(* CoDeSys 2.3 export: PALETIZER.EXP *)

(* Data type in EPT Lib/Achsen/BECKHOFF *)
TYPE struct_eccoe_sdo :
STRUCT
	s_ec_slave_net_id 		: T_AmsNetId := '';
	ui16_slave_addr 			: UINT := 0; (* Address of the slave device.*)
	i8_sub_index 				: BYTE := 0; (* CANopen Sdo subindex.*)
	w_index 					: WORD := 16#00; (* CANopen Sdo index.*)
	dw_p_source_buffer 		: DWORD := 16#0000; (* Contains the address of the buffer containing the data to be send. *)
	dw_p_destination_buffer	: DWORD := 16#0000; (* Contains the address of the buffer for the received data. *)
	ui32_buffer_length 			: UDINT := 0; (* Contains the max. number of bytes to be received. *)
	ui32_value 				: UDINT := 0; (* variable to be written to the CoE Object *)
	ui16_value 				: UINT := 0; (* variable to be written to the CoE Object *)
	byte_value 				: BYTE := 16#00; (* variable to be written to the CoE Object *)
	bool_value 				: BOOL := FALSE; (* variable to be written to the CoE Object *)
END_STRUCT
END_TYPE

(* Data type in EPT Lib/Achsen/EL72x1 *)
TYPE enum_ModeOfOperation :
	(
	CSP			:=	8,	(*cyclic synchronous position*)
	CSV			:=	9,	(*cyclic synchronous velocity*)
	CST			:=	10,	(*cyclic synchronous torque*)
	CSTCA		:=	11	(*cyclic synchronous torque with commutation angle*)
	);
END_TYPE

(* Data type in EPT Lib/Achsen/EL72x1 *)
TYPE st_config_axis :
STRUCT
	Description				:STRING;
	InstName				:STRING;
	Aktiv					:BOOL;
	Skalierfaktor				:LREAL;
	Bit_Geber				:INT;
	Getriebefaktor			:LREAL;
	Modulo					:BOOL:=TRUE;
	Pos_Faktor				:LREAL;						(*Weg bei einer Motorumdrehung in mm*)
	ModeOfOperation			:enum_ModeOfOperation:=CSP;
	maxRpm					:INT;				(*Maximale Drehzahl des Motor*)
(*nur für Coe-Online 7010.03 (CSP) position mode*)

	RampTime				:TIME;				(*Baustelle*)(*Beschleunigungszeit und Bremsrampe*)
	PosDiffControl_on			:BOOL;				(*Baustelle*)
	max_PosDiff				:LREAL;				(*Baustelle*)
	UeberlaufControl_on		:BOOL;
	Torque_Limit				:INT;				(*bei 0 ausgeschaltet*)(* Baustelle*)
	SW_Limit_on				:BOOL;
	SW_Limit_min			:LREAL;
	SW_Limit_max			:LREAL;
	lr_kp 					:LREAL := 800;
	lr_ki 						:LREAL := 100.0;
	lr_kd 					:LREAL := 50;
END_STRUCT
END_TYPE

(* Data type in EPT Lib/Achsen/EL72x1 *)
TYPE st_ctrl_Axis :
STRUCT
	in		: st_ctrl_in_axis;
	out		: st_ctrl_out_axis;
END_STRUCT
END_TYPE

(* Data type in EPT Lib/Achsen/EL72x1 *)
TYPE st_ctrl_in_axis :
STRUCT
	Position					:LREAL;

(*Bit 0*) Ready_to_switch_on	:BOOL;
(*Bit 1*) Switched_on			:BOOL;
(*Bit 2*) Operation_enabled		:BOOL;
(*Bit 3*) Fault					:BOOL;
(*Bit 4 : reserved*)
(*Bit 5 : reserved*)
(*Bit 6*) Switch_on_disabled		:BOOL;
(*Bit 7*) Warning				:BOOL;
(*Bit 8 + 9 : reserved*)
(*Bit 10*) TxPDOToggle		:BOOL; (*An-/Abwahl über 0x8010:01[} 136]*)
(*Bit 11*) Internal_Limit_active	:BOOL;
(*Bit 12*) Target_value_ignored	:BOOL;
(*Bit 13 - 15 : reserved*)

	Velocity				:LREAL;
	Following_Error		:LREAL;

END_STRUCT
END_TYPE

(* Data type in EPT Lib/Achsen/EL72x1 *)
TYPE st_ctrl_out_axis :
STRUCT
	Target_Position		:LREAL;
	Tearget_Velocity		:DINT;

(*Bit 0*)	Switch_on					:BOOL;
(*Bit 1*)	Enable_voltage		:BOOL;
(*Bit 2	*)Shutdown					:BOOL;
(*Bit 3*)	Enable_operation	:BOOL;
(*Bit 4 - 6 : reserved*)
(*Bit 7*)	Fault_reset				:BOOL;
(*Bit 8 - 15 : reserved*)

END_STRUCT
END_TYPE

(* Data type in EPT Lib/Achsen/EL72x1 *)
TYPE st_fb_axis :
STRUCT
	ton_uez			:TON;
	ton_uez_velo	:TON;
	ton_quitt		:TON;
	ton_aufPos		:TON;
	ton_Busy		:TON;


	r_trig_stop		: R_TRIG;
	r_trig_quitt	: R_TRIG;
	r_trig_reset	: R_TRIG;
	r_trig_jogP		: R_TRIG;
	r_trig_jogM		: R_TRIG;
	r_trig_MoveP	: R_TRIG;
	r_trig_MoveM	: R_TRIG;
	r_trig_MotorOn	: R_TRIG;
	r_trig_MoveAbs	: R_TRIG;

	r_trig_teach		: R_TRIG;
	r_trig_kont			: R_TRIG;
	r_trig_ink_10		: R_TRIG;
	r_trig_ink_100		: R_TRIG;
	r_trig_ink_1000		: R_TRIG;
	r_trig_ink_var		: R_TRIG;
	r_trig_Auto			: R_TRIG;
	r_trig_Hand			: R_TRIG;
END_STRUCT
END_TYPE

(* Data type in EPT Lib/Achsen/EL72x1 *)
TYPE st_Help_axis :
STRUCT
	b_init				:BOOL;
	b_init2				:BOOL;
	b_ToggleHelp		:BOOL;

	b_Pos_nr_Empty		:ARRAY [-1..NO_OF_POS_AXIS] OF BOOL;
	PosNr				:INT:=1;
	Pos					:LREAL;

END_STRUCT
END_TYPE

(* Data type in EPT Lib/Achsen/EL72x1 *)
TYPE st_PID_axis :
STRUCT
	lr_Override			:LREAL;

	lr_delta				: LREAL := 0.0;
	lr_delta_alt			: LREAL := 0.0;
	lr_delta_dif			: LREAL := 0.0;

	lr_current_p			: LREAL := 0.0;
	lr_current_i			: LREAL := 0.0;
	lr_current_d			: LREAL := 0.0;

	lr_current_v			: LREAL := 0.0;
	lr_tmp				: LREAL := 0.0;

	lr_delta_targetpos	: LREAL := 0.0;
	lr_targetpos_alt		: LREAL := 0.0;

END_STRUCT
END_TYPE

(* Data type in EPT Lib/Achsen/EL72x1 *)
TYPE st_Pos :
STRUCT
	Description		: STRING;
	Pos	 			: LREAL;
END_STRUCT
END_TYPE

(* Data type in EPT Lib/Achsen/EL72x1 *)
TYPE st_Pos_axis :
STRUCT
	ist					:REAL;
	soll					:REAL;
	r_18bit				:REAL;
	r_20bit				:REAL;
	r_32bit				:REAL;

	lr_DiffPuls			:LREAL := 0.0;
	lr_DiffVelo			:LREAL := 0.0;
	lr_MaxDiff			:LREAL := 0.0;

	(*Überlauf*)
	lr_akt_alt				:LREAL;
	lr_delta_ueberlauf		:LREAL;
	i32_count_ueberlauf	:DINT;
	lr_Uebrlauf_DistOne	:LREAL;
	lr_Uebrlauf_Dist		:LREAL;

	(*Singelturn*)
	lr_ModuloPosInc		:LREAL;
	lr_ModuloHelp		:LREAL;
	lr_ModuloHelp2		:LREAL;
	i16_ModuloHelp		:INT;
	lr_ModuloCount		:LREAL;

	(*Multiturn*)
	lr_Pos				:LREAL;
	lr_Target				:LREAL;
	lr_Mod				:LREAL;

	lr_Offset_Ink			:LREAL;
	i32_Offset_Ink			:UDINT;

END_STRUCT
END_TYPE

(* Data type in EPT Lib/Achsen/EL72x1 *)
TYPE st_sdo :
STRUCT
	fb_ec_coe_sdo_write_ex		: FB_EcCoESdoWriteEx;
	fb_ec_coe_sdo_read_ex		: FB_EcCoESdoReadEx;

(*	st_eccoe_sdo				:struct_eccoe_sdo;*)

	s_SlaveNetId 			: T_AmsNetId := '';
	ui16_SlaveAddr 			: UINT := 0;			 (* Address of the slave device.*)
	i8_SubIndex 			: BYTE := 0;			 (* CANopen Sdo subindex.*)
	w_Index 				: WORD := 16#00;	 (* CANopen Sdo index.*)

	acObjectData				:ARRAY[0..MAX_STRING_LENGTH] OF BYTE;

END_STRUCT
END_TYPE

(* Data type in EPT Lib/Achsen/EL72x1 *)
TYPE st_sm_axis :
STRUCT
	sm_timeout			:BOOL;
	sm_Error_Klemme	:BOOL;
	sm_Error_Warnung	:BOOL;
	sm_PosDiff			:BOOL;
	sm_Check_Velo		:BOOL;
	sm_SW_Limit			:BOOL;
	sm_fehler_daten_schreiben:BOOL;
	sm_connect			:BOOL;
	sm_Ueberlauf		:BOOL;
	sm_Torque_zu_gross	:BOOL;
	sm_NotausNok		:BOOL;
	sm_Move				:BOOL;
END_STRUCT
END_TYPE

(* Data type in EPT Lib/Achsen/EL72x1 *)
TYPE st_Velo_axis :
STRUCT
	maxRpmNachGertiebe	:LREAL;	(*Maximale Drehzahl nach Getriebe*)
	maxLinear		:LREAL;	(*Maximale Geschwindigkeit in mm/min*)
	maxRpm				:LREAL;	(*in U/min oder in mm/min*)
	Vorgabe_Velo_rpm	:LREAL;	(*in U/min*)
	sollRpm				:LREAL;	(*in U/min*)
	soll					:LREAL;
	ist				:LREAL;
	dif				:LREAL;
	Faktor			:LREAL;

END_STRUCT
END_TYPE

(* Data type in EPT Lib/Achsen/EL72x1 *)
TYPE st_Visu_axis :
STRUCT
	Einheit_pos			:STRING(10);
	Einheit_velo			:STRING(10);

	BtnReset			: sButtonVisu;
	BtnStop				: sButtonVisu;
	BtnJogP			: sButtonVisu;
	BtnJogM			: sButtonVisu;
	BtnMotorOn			: sButtonVisu;
	BtnMoveAbs		: sButtonVisu;
	BtnTeach			: sButtonVisu;

	PosNr				:INT:=1;
	Poslist				:BOOL;

	Control				:BOOL;
	b_kont				:BOOL;
	b_ink_10			:BOOL;		(*in µm*)
	b_ink_100			:BOOL;		(*in µm*)
	b_ink_1000			:BOOL;		(*in µm*)
	b_ink_var			:BOOL;		(*in mm variabel *)
	lr_ink_var			:LREAL:=10;

	b_Pos_nr			:ARRAY [-1..NO_OF_POS_AXIS] OF BOOL;
	b_PosNr			:BOOL;
END_STRUCT
END_TYPE

(* Data type in EPT Lib/Allgemeine Kontrollstrukturen Objekte *)
TYPE enum_step_nr :
	(
	INIT_OBJ := 0,
	INIT := 10,
	BEREIT := 100,
	HALT := 970,
	STOP := 980,
	FEHLER := 1000,
	INAKTIV:=2010
	);
END_TYPE

(* Data type in EPT Lib/Allgemeine Kontrollstrukturen Objekte *)
TYPE struct_config :
STRUCT
	str_instanz_name					: STRING(48) := '';
	str_beschreibung					: STRING(50) := '';
	b_station_aktiv					: BOOL := FALSE;
	b_station_in_simulation				: BOOL := FALSE;
	i16_meld_startindex				: INT := 0;
	b_config_fertig					: BOOL := FALSE;
END_STRUCT
END_TYPE

(* Data type in EPT Lib/Allgemeine Kontrollstrukturen Objekte *)
TYPE struct_ctrl :
STRUCT
	in		: struct_ctrl_in;
	out		: struct_ctrl_out;
END_STRUCT
END_TYPE

(* Data type in EPT Lib/Allgemeine Kontrollstrukturen Objekte *)
TYPE struct_ctrl_in :
STRUCT
	b_quitt						: BOOL := FALSE;
	b_stop 						: BOOL := FALSE;
         b_halt		  	 			: BOOL := FALSE;
         b_definierter_halt  	 			: BOOL := FALSE;
	b_init 						: BOOL := FALSE;
	b_init_2 						: BOOL := FALSE;
         b_preinit                				: BOOL := FALSE;
	b_start						: BOOL := FALSE;
	b_start_2						: BOOL := FALSE;
	b_gutteil_produziert 			: BOOL := FALSE;
	b_schlechtteil_produziert 		: BOOL := FALSE;
	b_start_lesen					: BOOL := FALSE;
	b_start_schreiben				: BOOL := FALSE;
	b_schutzhaube_ab			: BOOL := FALSE;
	b_schutzhaube_auf			: BOOL := FALSE;
	b_nachtabschaltung			: BOOL := FALSE;
	b_gehe_step_ibn				: BOOL := FALSE;
	b_ibn_start					: BOOL := FALSE;
	b_freigabe					: BOOL := FALSE;
END_STRUCT
END_TYPE

(* Data type in EPT Lib/Allgemeine Kontrollstrukturen Objekte *)
TYPE struct_ctrl_out :
STRUCT
	b_bereit 						: BOOL := FALSE;
	b_bereit_2					: BOOL := FALSE;
         b_prebereit               			: BOOL := FALSE;
	b_fehler 						: BOOL := FALSE;
	b_fertig						: BOOL := FALSE;
	b_fertig_2					: BOOL := FALSE;
	b_bandende					: BOOL := FALSE;
	b_kontroller_start				: BOOL := FALSE;
	b_gestoppt					: BOOL := FALSE;
	b_angehalten					: BOOL := FALSE;
	b_haube_oeffnen				: BOOL := FALSE;
	b_nachtabschaltung			: BOOL := FALSE;
	b_einzelfertigung				: BOOL := FALSE;
	b_busy						: BOOL := FALSE;
 st_takt_Time : STRING;
END_STRUCT
END_TYPE

(* Data type in EPT Lib/Allgemeine Kontrollstrukturen Objekte *)
TYPE struct_objekt :
STRUCT
	st_config		: struct_config;
	st_ctrl		: struct_ctrl;
END_STRUCT
END_TYPE

(* Data type in EPT Lib/Hydra *)
TYPE enum_StatusId :
	(

		(*
		M_S = Maschinenstörung,
		W_S = Werkzeugstörung,
		P_S = Peripheriestörung,
		AOI_S = Kamerastörung,
		M_W = Maschinenwartung,
		W_W = Werkzeugwartung,
		A_U = Ablaufunterbrechung
		*)


		_PRODUKTION := 1,
		_Nachtabschaltung_STOP := 199,
		_S_Quittiert := 290,
		_A_U_Steuerung_Aus := 299,
		_A_U_Auftrag_voll := 300,
		_M_S_Haube_Einzug := 301,
		_A_U_Trennstelle := 303,
		_A_U_Spule_voll := 304,
		_M_S_Haubenschaltleiste := 305,
		_M_S_Haube_Bandauslauf := 306,
		_M_S_Klappe_hinten := 307,
		_M_S_Klappe_links := 308,
		_M_S_Klappe_rechts := 309,
		_M_S_Klappe_vorne := 310,
		_M_S_Temp_Schaltschrank := 311,
		_M_S_Temp_Haubenmotor := 312,
		_M_S_Temp_Haubenluefter := 313,
		_M_S_Bandoeler_Fuellstand := 314,
		_M_S_Bandoeler := 315,
		_M_W_Pressenkopf := 316,
		_M_W_Zahnriemen := 317,
		_M_W_Wartungseinheit := 318,
		_M_W_Bandeinzug := 319,
		_M_W_Werkzeug := 320,
		_M_S_Drehgeber := 321,
		_M_S_Hauptantriebsmotor := 322,
		_M_S_Abfallbehaelter := 323,
		_W_S_Bandaufgestellt := 325,
		_W_S_Parallelschnitt := 326,
		_W_S_Gesamtschnitt_o := 327,
		_W_S_Gesamtschnitt_u := 328,
		_W_S_Dyn_Schnittueberw_eins := 329,
		_W_S_Dyn_Schnittueberw_zwei := 331,
		_W_S_Faengerueberw_eins := 332,
		_W_S_Faengerueberw_zwei := 333,
		_W_S_Faengerueberw_drei := 334,
		_W_S_Faengerueberw_vier := 335,
		_W_S_Position_Wkz := 336,
		_W_S_Pfostenabfrage := 337,
		_W_S_Tcom_eins := 338,
		_W_S_Tcom_zwei := 339,
		_W_S_Bandschneideueberwachung := 340,
		_W_S_Pinabstanzueberwachung := 341,
		_AOI_S_Kamera :=343,
		_P_S_Aufhaspel := 350,
		_P_S_Abhaspel := 351,
		_M_S_Not_Halt := 352,
		_M_S_Auffahrsicherung := 353,
		_Trennstelle := 809,
		_Maschine_STOP :=843,
		_Peripherie_STOP := 844,
		_Stoerung_Lasertriangulation := 870,
		_Stoerung_Bsh_Zellen := 871,
		_Maschinenstoerung := 884,
		_Peripheriestoerung := 885,
		_WERKZEUGSTOERUNG := 886,
		 _Kamerastoerung := 887,
		_HV_Stoerung := 888,
		_Schichtfrei := 999

);

END_TYPE

(* Data type in EPT Lib/Hydra *)
TYPE struct_Hydra :
STRUCT
	s_Start_Time	: STRING(20) := '01.01.1970 00:00:00';	(* TT.MM.JJJJ HH:MM:SS *)
	i_Counter		: ARRAY[1..104] OF DINT;	(* alle Zähler 4-stellig *)
	b_Input		: ARRAY[1..128] OF BOOL:=128(FALSE);
END_STRUCT
END_TYPE

(* Data type in EPT Lib/Hydra *)
TYPE struct_Hydra8 :
STRUCT
	iCounter		: ARRAY[1..20] OF DINT;	(* alle Zähler 4-stellig *)
	bStatus		: ARRAY[1..999] OF BOOL:=999(FALSE);	(* TRUE wenn Status aktiv ist *)
END_STRUCT
END_TYPE

(* Data type in EPT Lib/sDatensatz/sTypeDaten *)
TYPE sData_b :
STRUCT

	Description					: STRING(50); 	(* Beschreibung *)
	b								: BOOL; 		(* Wert *)

END_STRUCT
END_TYPE

(* Data type in EPT Lib/sDatensatz/sTypeDaten *)
TYPE sData_byte :
STRUCT

	Description					: STRING(50); 	(* Beschreibung *)
	BYT								: BYTE; 			(* Wert *)
	Unit				   			: STRING(20);	(* Einheit *)

END_STRUCT
END_TYPE

(* Data type in EPT Lib/sDatensatz/sTypeDaten *)
TYPE sData_i16 :
STRUCT

	Description					: STRING(50); 	(* Beschreibung *)
	i16								: INT; 			(* Wert *)
	Unit				   			: STRING(20);	(* Einheit *)

END_STRUCT
END_TYPE

(* Data type in EPT Lib/sDatensatz/sTypeDaten *)
TYPE sData_i32 :
STRUCT

	Description		: STRING(50); 	(* Beschreibung *)
	i32					: DINT; 		(* Wert *)
	Unit				: STRING(20);	(* Einheit *)

END_STRUCT
END_TYPE

(* Data type in EPT Lib/sDatensatz/sTypeDaten *)
TYPE sData_lr :
STRUCT

	Description		: STRING(50); 	(* Beschreibung *)
	lr					: LREAL; 			(* Wert *)
	Unit		   		: STRING(20);	 	(* Einheit *)

END_STRUCT
END_TYPE

(* Data type in EPT Lib/sDatensatz/sTypeDaten *)
TYPE sData_Str :
STRUCT

	Description				: STRING(50); 	(* Beschreibung *)
	str							: STRING(50); 	(* Text *)

END_STRUCT
END_TYPE

(* Data type in EPT Lib/sDatensatz/sTypeDaten *)
TYPE sData_ui32 :
STRUCT

	Description			: STRING(50); 	(* Beschreibung *)
	i32						: UDINT; 		(* Wert *)
	Unit					: STRING(20);	(* Einheit *)

END_STRUCT
END_TYPE

(* Data type in sStation/MainMenue *)
TYPE sMainMenue:
STRUCT
	BtnMainMenue					:sButtonVisu_Tree;
	BtnManual						:sButtonVisu_Tree;
	BtnManual_ST00_0				:sButtonVisu_Tree;	(*Allgemein*)
		BtnManual_ST00_1			:sButtonVisu_Tree;	(*Türen und Not-Halt*)
		BtnManual_ST00_2			:sButtonVisu_Tree;	(*Flügelkamera*)
	BtnManual_ST02_0				:sButtonVisu_Tree;	(*Rundtisch*)
	BtnManual_ST03_0				:sButtonVisu_Tree;	(*Roboter*)
			BtnManual_ST03_xx		:sButtonVisu_Tree;	(*Rüstsatz Seite1*)
			BtnManual_ST03_xx_2	:sButtonVisu_Tree;	(*Rüstsatz Seite2*)
	BtnManual_ST08_0				:sButtonVisu_Tree;
		BtnManual_ST08_1			:sButtonVisu_Tree;	(*Blisterzuführung*)
		BtnManual_ST08_2			:sButtonVisu_Tree;	(*Abstapeln*)
		BtnManual_ST08_3			:sButtonVisu_Tree;	(*Bandstrecke*)
		BtnManual_ST08_4			:sButtonVisu_Tree;	(*Aufstapeln*)


	BtnTD							:sButtonVisu_Tree;
	BtnTD01_Edit					:sButtonVisu_Tree;
	BtnTD02_Edit					:sButtonVisu_Tree;

	BtnMP_Main					:sButtonVisu_Tree;
	BtnMP_ST1						:sButtonVisu_Tree;
	BtnMP_ST2						:sButtonVisu_Tree;
	BtnMP_Date					:sButtonVisu_Tree;
	BtnMP_Service					:sButtonVisu_Tree;

	BtnSystem						:sButtonVisu_Tree;
		Btn_ErrorLog				:sButtonVisu_Tree;
		Btn_ErrorList				:sButtonVisu_Tree;
		Btn_Gst						:sButtonVisu_Tree;
		Btn_Step_Diag				:sButtonVisu_Tree;
		Btn_Lng					:sButtonVisu_Tree;

		Btn_VisuBeenden			:sButtonVisu_Tree;
END_STRUCT
END_TYPE

(* Data type in sStation/sMachineParameter/Service *)
TYPE eService_Type :
	(
	BETRIEBSSTUNDEN			:=	0,
	STUNDEN			:=	1,
	TAGE				:=	2,
	COUNTER			:=	3
	);
END_TYPE

(* Data type in sStation/sMachineParameter/Service *)
TYPE sMachParaService :
STRUCT
	visu			: ARRAY[0..15] OF struct_visu_service;
	daten			: ARRAY[0..15] OF struct_daten_service;
	betriebssekundenzaehler	:UDINT;
END_STRUCT
END_TYPE

(* Data type in sStation/sMachineParameter/Service *)
TYPE struct_daten_service :
STRUCT
	Name			: STRING(255);
	Default_Value	: LREAL;
	Current_Value	: LREAL;
	Warning_Value	: LREAL;
	Warning_reached	: BOOL:= FALSE;
	Default_reached	: BOOL:= FALSE;
	Type_Service	: eService_Type;
	Unit				: STRING(20);
	Starttag			: INT := 0;
	Startstunden	: LREAL := 0;
	StartBetriebsStd	: LREAL := 0;
END_STRUCT
END_TYPE

(* Data type in sStation/sMachineParameter/Service *)
TYPE struct_visu_service :
STRUCT
	BtnReset			: sButtonVisu;
	BtnStart			: sButtonVisu;
	BtnType			: sButtonVisu;
	Current_Value	 : STRING(20);
	Current_Value_Color	: DINT;

END_STRUCT
END_TYPE

(* Data type in sStation/sMachineParameter *)
TYPE sMachineParameterHandling :
STRUCT
(* ST01 *)
	Dummy:BOOL;
(* ST02 *)

(* ST03 *)

(* ST04 *)

(* ST05 *)
END_STRUCT
END_TYPE

(* Data type in sStation/sMachineParameter *)
TYPE sMachPara :
STRUCT
	sLastTDfile							: STRING;
	ShiftData							: sMP_ShiftHandler;
	ST00: sMachParaST00; (*Instancename is Filename in Typedata Folder*)
	ST02: sMachParaST02; (*Instancename is Filename in Typedata Folder*)
	ST03: sMachParaST03; (*Instancename is Filename in Typedata Folder*)
	ST08: sMachParaST08; (*Instancename is Filename in Typedata Folder*)
	Visu:	sMachineParameterHandling; (* Object Collection for Parameterhandling in Visu - e.g. Buttons - Called in System/VisuInterface/MachParaHandling  *)
END_STRUCT
END_TYPE

(* Data type in sStation/sMachineParameter *)
TYPE sMachParaST00 :
STRUCT
	Override					:	DINT :=10;
	OverrideForHoming	:	DINT :=5;
	MaxLogInTime				: DINT  := 0;
	Sprache    					: STRING(10);

	ActPartNo			: DINT; (*laufende Nr. für Laser-String*)

	IFMCameraActive			: BOOL := TRUE;
	IFMCameraActiveText		:STRING :='ON';

	Cam_NoOfErrors		: DINT := 1;

(* -----------------------------------------------------------------------------------------
		Sollwerte
  ----------------------------------------------------------------------------------------- *)

	PartsToProduce					: DINT;		(* Sollstückzahl *)
	PartsToProduceOffset		: DINT;		(* Korrenkturwert auf Sollstückzahl *)

 	PartsNokInSeriesAllowed : DINT := 0;		(* max. Fehler in Folge *)

	PartsNokPerSubset				: DINT :=0;		(* max. erlaubete n.i.O. Teileanzahl pro Untermenge *)
	PartsNokSubsetSize			: DINT :=100;		(* Untermengengröße *)

(* -----------------------------------------------------------------------------------------
		Istwerte
  ----------------------------------------------------------------------------------------- *)

	PartsInserted						: DINT;		(* Teile aufgesetzt in ST01 *)
	PartsNokTotal						: DINT;		(* Teile n.i.O. gesamt *)
	PartsOkTotal						: DINT;		(* Teile i.O. gesamt, eingesetzt in Blister/Tube *)
	PartsRemaining					: DINT;		(* Teile noch zu produzieren (PartsToProduce + PartsToProduceOffset + PartsNokTotal - PartsInserted) *)

	PartsNokTotalNoReset		: DINT;		(* Teile n.i.O. gesamt *)
	PartsOkTotalNoReset			: DINT;		(* Teile i.O. gesamt, eingesetzt in Blister/Tube *)

	LAN_no						: sData_i16:=(Description:='LAN_no', Unit:='no');
END_STRUCT
END_TYPE

(* Data type in sStation/sMachineParameter *)
TYPE sMachParaST02 :
STRUCT
	Override_Band				:	DINT :=10;

	RunTableEmpty 			: DINT := 5; (*Time in sec. *)
	IFMPos					: LREAL;
	IFMPosDummy			: LREAL;
	TableData				: ARRAY [1..NO_OF_NEST] OF sStationData;
	CamOn					: BOOL;
	CamNoOfErrors			: DINT := 1;
	CamNoOfErrorsPercent	: DINT := 1;
	DummyPruefung_93pol	: BOOL;
  	Dummy_test_Result  	: ARRAY [1..12] OF BOOL;
	NoOfDummys			: DINT := 6;
	SensopartIPAdress		: STRING(15);
	SensopartIPAdress2		: STRING(15);
	SensopartEthernet		: BOOL;

END_STRUCT
END_TYPE

(* Data type in sStation/sMachineParameter *)
TYPE sMachParaST03 :
STRUCT

	WpcInStackFilled		: BOOL;

	ActualPartsInPallet 		: DINT; (* Counter *)

	NoOfBlisterInStackerOut	: DINT; (* Counter *)

	ActualPartsOnBuffer 		: DINT; (* Counter *)

	ResetBuffer             : BOOL;
	(* Inputvariablen *)
	PartsInPallet	      	   : DINT; (* Max No Of Parts in Buffer *)

	NoOfTestParts				:	DINT;

	FrontCamOn			: BOOL;
	BackCamOn			: BOOL;
	CamNoOfErrors			: DINT := 1;
	CamNoOfErrorsPercent	: DINT := 1;

	RobotIPAdress			: STRING(15);
	BandMoveP				:BOOL;
	SGM_3621		: BOOL;

	BeltMotorCheckPartActive          : BOOL;

	RoboterColisionActivated	 :BOOL;

	CamOn					: ARRAY [1..2] OF BOOL;		(*Sensopart Kamera*)
	SensopartIPAdress		: ARRAY [1..2] OF STRING(15);

	CamOn_KYE				: BOOL;			(*Keyence Kamera*)
	CamNoOfErrors_KYE		: DINT := 1;
	CamNoOfErrorsPercent_KYE: DINT := 1;

END_STRUCT
END_TYPE

(* Data type in sStation/sMachineParameter *)
TYPE sMachParaST08 :
STRUCT
	NoOfBlisterInStackerOut			: DINT; (* Counter *)

	StapelMotor								: BOOL;
	PosOffsetAufstapeln	 			: st_Pos;
	PosOffsetAbstapeln	 			: st_Pos;
	Override_Aufstapeln				: DINT :=10;
	Override_Abstapeln				: DINT :=10;
	Traystapel_schieben 			: BOOL:=TRUE;
	Trayzufuhr_Verlaengerung		: BOOL:=TRUE;
	TrayAushebenMotor				: BOOL;
	PosOffsetTrayAusheben 			: st_Pos;
	Override_TrayAusheben			: DINT :=10;

END_STRUCT
END_TYPE

(* Data type in sStation/sPersistent *)
TYPE sPersDaten :
STRUCT

	i_DayOfYearAutoCheckIn	:DINT;

END_STRUCT
END_TYPE

(* Data type in sStation/sTurnTable *)
TYPE sProcessData :
STRUCT

	Nest_Nr			: DINT;
	Part				: BOOL;
	Result 			: DINT;					(*   0 = Teil noch nicht bearbeitet bzw. Nest leer*)
											(*   1 =  Oberseite OK*)
											(*  11 = Oberseite und Unterseite OK*)
											(*  99 = Teil ist NOK	*)
END_STRUCT
END_TYPE

(* Data type in sStation/sTurnTable *)
TYPE sStationData :
STRUCT
	Description				: STRING:='';
	HomePos				: BOOL;
	Activated				: BOOL := TRUE; (* Station Deactivated *)
	CycleTime				: DINT;

	ProcessData			: sProcessData; (*is shifted when Table turns*)
END_STRUCT
END_TYPE

(* Data type in sStation/sTypedata *)
TYPE sTypeData :
STRUCT
	(* allegmeine Typinfos *)
	ArtNo					: STRING(30); (* interne Kundenartikelnummer *)
	TypeName				: STRING(30); (* xml-Dateiname *)
	TypeDescription			: STRING(30); (* Typbeschreibung optional *)

	(* Typmerkmale *)
	TypeCode				: STRING(5); (* Typkennung z.B. P310 *)

	Override_Band			: INT:=20; (* *)
	Override_Robi			: INT:=20; (* *)

	PosAbstapeln	 		: ARRAY [1..NO_OF_POS_AXIS] OF st_Pos;	(*	1=unten, 2= mitte, 3=oben*)
	PosAufstapeln	 		: ARRAY [1..NO_OF_POS_AXIS] OF st_Pos;	(*	1=unten, 2= mitte, 3=oben*)
	PosTrayAusheben	 		: ARRAY [1..NO_OF_POS_AXIS] OF st_Pos;	(*	1=unten, 2=oben*)

	TestpartBilister		: BOOL;
	DistIso					: LREAL;

	IFM_Positon_Dummy 		: LREAL ;
	SensopartErgebnis			: STRING(15); (*Ergebnis Sensopart Kamera*)
	Sensopart2Ergebnis			: STRING(15); (*Ergebnis Sensopart Kamera*)
	NoOfPalletsPerStack		: DINT:=1;

	(*Aus Load Info*)
	RobotOffset				: DINT;

	PartsInBlisterInlet		: DINT; (* Anzahl Teile pro Blister Einlauf *)
	PartsInRoboGripper		: DINT:=1; (* Anzahl Teile pro Robi Greifer *)

	IFM_CamProgNo			: BYTE;
	Sensopart_CamProgNo		: BYTE;
	Sensopart2_CamProgNo		: BYTE;
	Keyence_CamProgNo		: BYTE;

END_STRUCT
END_TYPE

(* Data type in sStation/sUserList *)
TYPE sUserList :
STRUCT
  	UserList							:	ARRAY [1..NO_OF_USERS] OF sUserData;
END_STRUCT
END_TYPE

(* Data type in sStation/sVisuInterface *)
TYPE sVisu:
STRUCT
(*---------------------------------------------------------------------------
  System
  ---------------------------------------------------------------------------*)
	ErrorHandler				: sErrorHandlerVisu;
	ErrorHistory				: sErrorHandlerVisu;
	ErrorHistoryScroll		: DINT;
	SelectPictureName		: STRING(20);
	SavePersistentData  	: BOOL;

	Message				: sMessageVisu;
	ModeSelect				: sModeSelectVisu;
	LoginHandler			: sVisuLoginDialog;
	MainMenue				: sMainMenue;

(*---------------------------------------------------------------------------
  Station00
  ---------------------------------------------------------------------------*)
	ST00_40_F1 			: sDigInVisu; (* Vorsicherungen Leistung iO *)
	ST03_210_S1 			: sDigInVisu; (* Not-Aus 1 Anlage ausgelöst *)
	ST08_210_S2 			: sDigInVisu; (* Not-Aus 2 Anlage ausgelöst *)
	ST00_X4_16	 		: sDigInVisu; (* Not-Halt 2 Tampondrucker ausgelöst *)
	ST00_200_A1_A1 		: sDigInVisu; (* Not-Aus iO *)
	ST00_220_S1	 		: sDigInVisu; (* Schutztüre 1 geöffnet *)
	ST00_220_S2	 		: sDigInVisu; (* Schutztüre 1 geöffnet *)
	ST00_230_S2_E1 		: sDigInVisu; (* Schutztüre 1 geschlossen *)
	ST00_240_S1 		: sDigInVisu; (* Schutztüre 9 geschlossen *)
	ST00_226_S1			: sDigInVisu;(*Hubtüre 1 Schleuse Einlauf STN 8 geschlossen*)
	ST00_226_S2			: sDigInVisu;(*Hubtüre 2 Schleuse Einlauf STN 8 geschlossen*)
	ST00_227_S1			: sDigInVisu;(*Hubtüre 3 Schleuse Auslauf STN 8 geschlossen*)
	ST00_227_S2			: sDigInVisu;(*Hubtüre 4 Schleuse Auslauf STN 8 geschlossen*)
	ST00_229_S1			: sDigInVisu;(*Schutztüre Einlauf Tray STN 8 geschlossen*)
	ST00_230_S1			: sDigInVisu;(*Schutztüre Auslauf Tray STN 8 geschlossen*)
	ST00_231_S1			: sDigInVisu;(*Schutztüre Panel / Rutsche STN 8 geschlossen*)
	ST00_232_S1			: sDigInVisu;(*Schutztüre 8 Auslauf Tray STN 8 geschlossen*)
	ST00_170_Motorschutz	: sDigInVisu;(*Motorschutz in Ordnung*)
	ST00_170_Thermokont	: sDigInVisu;(*Thermokontakt in Ordnung*)
	ST00_228_S1      		 : sDigInVisu;
	ST00_71_X1_3  		: sDigInVisu; (* Schnittstelle Bedrucken Tinte JSK auf Übergabeposition *)
	ST00_71_X1_4  		: sDigInVisu; (* Schnittstelle Bedrucken Tinte Druckstation betriebsbereit *)
	ST00_72_X1_3  		: sDigInVisu; (* Schnittstelle Tampondrucker Teil in Abholposition *)(*Band Entnahmeposition 1*)
	ST00_72_X1_8  		: sDigInVisu; (* Schnittstelle Tampondrucker Druck abgeschlossen *)
	ST00_292_S1_STOP 	: sDigInVisu; (* Bedienstelle Produktion Stop *)
	ST00_292_S2_START	: sDigInVisu; (* Bedienstelle Produktion Start *)
	ST00_292_S3_RESET	: sDigInVisu; (* Bedienstelle Produktion Reset *)
	ST00_350_B20_0 		: sDigInVisu; (* Druckschalter Wartungseinheit Hauptluft min.6 bar *)

	ST00_245_V1			: sDigOutInVisu; (* Verriegelung Schutztüren-Leuchte *)
	ST00_245_V2_START	: sDigOutInVisu; (* Bedienstelle Start-Leuchte *)
	ST00_245_V3_RESET	: sDigOutInVisu; (* Bedienstelle Reset-Schutztüren-Leuchte *)
	ST00_245_S1_STOP 	: sDigInVisu;	 (* Bedienstelle Produktion Stop *)
	ST00_245_S2_START	: sDigInVisu;	 (* Bedienstelle Produktion Start *)
	ST00_245_S3_RESET	: sDigInVisu;	 (* Bedienstelle Produktion Reset *)

	ST00_31_K1 			: sDigOutInVisu; (* Beleuchtung Anlage *)
	ST00_350_H1 			: sDigOutInVisu; (* Signalsäule RD Maschine Alarm/Störung *)
	ST00_350_H2 			: sDigOutInVisu; (* Signalsäule YE Bedienereingriff erforderlich *)
	ST00_350_H3 			: sDigOutInVisu; (* Signalsäule GN Maschine Automatik *)
	ST00_200_A1_E4 		: sDigOutInVisu; (* Quittierung Not-Aus *)
	ST00_220_S1_S31 		: sDigOutInVisu; (* Verriegelung Schutztüren *)
	ST00_292_H2_START	: sDigOutInVisu; (* Bedienstelle Start-Leuchte *)
	ST00_292_H3_RESET	: sDigOutInVisu; (* Bedienstelle Reset-Leuchte *)

	ST00_71_K2	  		: sDigOutInVisu; (* Schnittstelle Bedrucken Tinte Abholposition frei *)

	ST00_73_K2	  		: sDigOutInVisu; (* Schnittstelle allgemein Störung Tampondrucker *)
	ST00_73_K3	  		: sDigOutInVisu; (*Schnittstelle Förderband frei für Spritzmaschine*)
	ST00_73_K4	 		: sDigInVisu; 	(*Schnittstelle Freigabe von Spritzmaschine (nur für Anlagen ohne Rundtisch) *)


	ST00_74_Y2_4 : sValveVisu; (*ST00_74_Y2_4 Stopper Bandstrecke (Valve) *)
	ST00_74_Y2_5 : sValveVisu; (*ST00_74_Y2_5 Vereinzeler Bandstrecke (Valve) *)

	ST03_65_Q1			: sDigOutInVisu;		(* Kühltunnel (Lüfter)*)
	ST03_65_F1			: sDigInVisu;			(* Sicherung Kühltunnel (Lüfter)*)

(*---------------------------------------------------------------------------
  Station02
  ---------------------------------------------------------------------------*)
	ST02_FDB_55X1_5_READY 	:sDigInVisu; (* IFM Kamera Flügelerkennung links Ready *)
	ST02_FDB_55X1_6_IO			:sDigInVisu; (* IFM Kamera Flügelerkennung links Ergebnis iO *)
	ST02_FDB_55X1_6_NIO		:sDigInVisu; (* IFM Kamera Flügelerkennung links Ergebnis niO *)
	ST02_FDB_55X1_2_TRIGGER 	:sDigOutInVisu; (* IFM Kamera Flügelerkennung links Trigger *)
	ST02_FDB_55X1_7_JOB_BIT1 	:sDigOutInVisu;(* IFM Kamera links  Jobwechsel Bit 1 *)
	ST02_FDB_55X1_7_JOB_BIT2 	:sDigOutInVisu;(* IFM Kamera links  Jobwechsel Bit 2 *)

	ST02_FDB_56X1_5_READY 	:sDigInVisu; (* IFM Kamera Flügelerkennung rechts Ready *)
	ST02_FDB_56X1_6_IO			:sDigInVisu; (* IFM Kamera Flügelerkennung rechts Ergebnis iO *)
	ST02_FDB_56X1_6_NIO		:sDigInVisu; (* IFM Kamera Flügelerkennung rechts Ergebnis niO *)
	ST02_FDB_56X1_2_TRIGGER 	:sDigOutInVisu; (* IFM Kamera Flügelerkennung rechts Trigger *)
	ST02_FDB_56X1_7_JOB_BIT1 	:sDigOutInVisu;(* IFM Kamera links  Jobwechsel Bit 1 *)
	ST02_FDB_56X1_7_JOB_BIT2 	:sDigOutInVisu;(* IFM Kamera links  Jobwechsel Bit 2 *)

	ST02_S1_70K61_A1	:sDigOutInVisu; 	(* Start  Bedrucken *)

	ST02_S1_40K01 		:sDigInVisu;			(*  Freigabe Förderband von SPM *)
	ST02_FDB_80_B02 		:sDigInVisu;			(*  Band Entnahmeposition 2*)
	ST02_35_S31			:sDigInVisu; 			(* ST02 Druckschalter Wartungseinheit Hauptluft min.6 bar *)
	ST02_S1_6A01 			:sDigInVisu; 			(* ST02 Sicherung 24V *)

	ST02_FDB_40_B61	:sDigInVisu; 			(* Iso von SPM auf Band abgelegt *)
	ST02_FDB_40_B71	:sDigInVisu; 			(* Iso auf Band vor Vereinzler *)

	ST02_62_Y6			:sValveVisu; 			(*Tisch drehen 0 - 180 Grad (Valve) *)
	ST02_62_Y9			:sValveVisu; 			(*Schwenkarm 2 drehen 90 - 180 Grad (Valve) *)
	ST02_62_Y11			:sValveVisu; 			(* Schwenkarm 2 drehen 90 - 0 Grad (Valve) *)
	ST02_62_Y13			:sValveVisu; 			(*Schwenkarm 1 drehen 90 - 180 Grad (Valve) *)
	ST02_62_Y15			:sValveVisu; 			(*Schwenkarm 1 drehen 90 - 0 Grad (Valve) *)
	ST02_62_Y17			:sValveVisu; 			(*Schwenkarm 1 ISK Fixierung ein/ausfahren(Valve) *)
	ST02_62_Y18			:sValveVisu; 			(*Schwenkarm 2 ISK Fixierung ein/ausfahren(Valve) *)
	ST02_62V1				:sValveVisu; 			(* ISK Stopper ein-/ausfahren*)
	ST02_62V2				:sValveVisu; 			(* ISK Vereinzeler ein-/ausfahren*)
	ST02_62_Y4   			:sValveVisu; 			(*ST02_62_Y4 Kamera Ausschleusen Bandstrecke (Valve) *)

	ST02_35Y01 			:sValveVisu; 			(*1: Einschaltventil Hauptluft Tampondruckanlage*)

	ST02_FDB_54_B41		:sDigInVisu; (* Kamera ISK anwesend an Prüfposition *)

	ST02_DT_65B11  		:sDigInVisu; (* Tampondrucker Nest 1 leer *)
	ST02_DT_65B21  		:sDigInVisu; (* Tampondrucker Nest 2 leer *)

	ST03_51_M1 			: sDigInVisu; (* Bandmotor *)
	ST03_60_M1 			: sDigInVisu; (* Bandmotor Prüfteile *)


(*---------------------------------------------------------------------------
  Station03
  ---------------------------------------------------------------------------*)
	ST03_125_F1 		: sDigInVisu; (* Absicherung Roboter iO *)
	Robot01					:	sEpsonRobotVisu;

	St03_120_A1_A14: sDigInVisu;(*Roboter opt.- Tool 2 ist ein*)
	ST03_400_B12_6 : sDigInVisu; (* Schwenkmodul AST (Roboterkopf) *)
	ST03_400_B12_7 : sDigInVisu; (* Schwenkmodul GST (Roboterkopf) *)
	ST03_400_B54_7: sDigInVisu; (* Tray Testteile in Position *)
	ST03_8_75_B13_5: sDigInVisu; (*voll/belegt keine Prüfmittel mehr*)
	ST03_8_75_B13_6: sDigInVisu; (*belegt mit 6 Prüfmittel*)
	ST03_BG3_X53_0:	sDigOutInVisu; (*Taster Start Band Dummyprüfung*)
	ST03_A5 : sDigOutInVisu; (* Förderbandmotor Oriental *)
	ST03_601V1_A1 : sDigOutInVisu; (* FörderbandPrüfteile *)
	ST03_V2	: sDigInVisu; (* Störung Motor Förderband Oriental *)

	(*Rüstsatz 154 Rasterplattel*)
	ST03_418_B60_6: sDigInVisu;		(*  Zuführung links frei zum Ablegen ISK SP Maschine *)
	ST03_418_B60_7: sDigInVisu;		(*  Zuführung rechts frei zum Ablegen ISK SP Maschine *)

	ST03_419_B61_0: sDigInVisu;		(*  Förderband Zuführung links ISK anwesend zum Vereinzeln*)
	ST03_419_B61_1: sDigInVisu;		(*  Förderband Zuführung rechts ISK anwesend zum Vereinzeln*)
	ST03_419_B61_2: sDigInVisu;		(*  Züführung links ISK auf Übergabeposition Roboter Palettierer*)
	ST03_419_B61_3: sDigInVisu;		(*  Züführung rechts ISK auf Übergabeposition Roboter Palettierer*)

	ST03_419_Y61_5 : sValveVisu; 		(* Förderband linke Zuführung Vereinzler AST/GST *)
	ST03_419_Y61_6 : sValveVisu; 		(* Förderband rechte Zuführung Vereinzler AST/GST *)
	ST03_419_Y61_7 : sValveVisu; 		(* Förderband links/rechts Züführung Stopper AST/GST *)

	(*Rüstsatz 154pol*)

	ST03_425_B67_4: sDigInVisu;		(*  Zuführung  frei zum Ablegen ISK SP Maschine Pos.1 *)
	ST03_425_B67_5: sDigInVisu;		(*  Zuführung  frei zum Ablegen ISK SP Maschine Pos.2 *)
	ST03_425_B67_6: sDigInVisu;		(*  Zuführung  frei zum Ablegen ISK SP Maschine Pos.3 *)
	ST03_425_B67_7: sDigInVisu;		(*  ISK anwesend am Vereinzler*)

	ST03_426_B68_4: sDigInVisu;		(*  Züführung  ISK auf Übergabeposition Roboter Palettierer*)
	ST03_426_Y68_5 : sValveVisu; 		(* Förderband  Zuführung Vereinzler AST/GST *)
	ST03_426_Y68_6 : sValveVisu; 		(* Förderband  Züführung Stopper AST/GST *)


	(*Rüstsatz 160pol*)
	ST03_421_B63_4: sDigInVisu;		(*  Förderband frei zum Ablegen ISK SP Maschine Pos1 *)
	ST03_421_B63_5: sDigInVisu;		(*  Förderband frei zum Ablegen ISK SP Maschine Pos2 *)
	ST03_421_B63_6: sDigInVisu;		(*  Förderband frei zum Ablegen ISK SP Maschine Pos3 *)
	ST03_421_B63_7: sDigInVisu;		(*  ISK anwesend am Vereinzler*)
	ST03_422_B64_0: sDigInVisu;		(* Förderband Trigger Tintenstrahldrucker 1 (Lichtschranke)Rüstsatz*)
	ST03_423_B66_0: sDigInVisu;		(* Förderband Trigger Tintenstrahldrucker 2 (Lichtschranke) Rüstsatz*)
	ST03_8_B76_1: sDigInVisu;		(* Förderband Trigger Tintenstrahldrucker (Lichtschranke) 3621*)
	ST03_8_B76_2: sDigInVisu;		(* Förderband Trigger Tintenstrahldrucker (Lichtschranke) 3621*)
	ST03_422_B64_3: sDigInVisu;		(* Förderband ISK anwesend Stopper 1 Kamera*)
	ST03_423_B65_2: sDigInVisu;		(* Förderband ISK anwesend Stopper 2 Kamera*)
	ST03_423_B65_5: sDigInVisu;		(* Förderband ISK anwesend Stopper 3 Kamera*)
	ST03_422_B64_4: sDigInVisu; 		(* Zuführung ISK auf Übergabeposition Robo Palettierer*)

	ST03_422_Y64_5 : sValveVisu; 		(* Förderband  Zuführung Vereinzler AST/GST *)
	ST03_422_Y64_6 : sValveVisu; 		(* Förderband  Stopper Vereinzler AST/GST *)
	ST03_422_Y64_7 : sValveVisu; 		(* Förderband  Stopper 1 Kamera AST/GST *)
	ST03_423_Y65_6 : sValveVisu; 		(* Förderband  Stopper 2 Kamera AST/GST *)
	ST03_423_Y65_7 : sValveVisu; 		(* Förderband  Stopper 3 Kamera AST/GST *)

	ST03_33F4: sDigInVisu; 			(*Steckdosenleise Tintenstrahldrucker*)
	ST03_70U3_1: sDigInVisu; 			(*Bereit/ Im Druck Tintenstrahldrucker Frontseite*)
	ST03_70U3_2: sDigInVisu; 			(*Tank voll Tintenstrahldrucker Frontseite*)
	ST03_70U3_3: sDigInVisu; 			(*Fehler/Störung Tintenstrahldrucker Frontseite*)
	ST03_71U3_1: sDigInVisu; 			(*Bereit/ Im Druck Tintenstrahldrucker Rückseite*)
	ST03_71U3_2: sDigInVisu; 			(*Tank voll Tintenstrahldrucker Rückseite*)
	ST03_71U3_3: sDigInVisu; 			(*Fehler/Störung Tintenstrahldrucker Rückseite*)

	ST03_PLAN_70V1_1:sDigOutInVisu; 	(* Start  Bedrucken Tintenstrahldrucker Frontseite*)
	ST03_PLAN_71V1_2:sDigOutInVisu; 	(* Start  Bedrucken Tintenstrahldrucker Rückseite*)

	ST03_Y01 			: sValveVisu; 			(*1: Einschaltventil Hauptluft Tintenstrahldrucker nur bei SG-Maschine 3621*)
	ST03_S18			: sDigInVisu; 			(* ST02 Druckschalter Wartungseinheit Hauptluft min.6 bar *)
	ST03_H6 			: sDigOutInVisu; 		(* Signalsäule GR Bedruckung IO *)
	ST03_H7 			: sDigOutInVisu; 		(* Signalsäule RD Sammelstörung Bedruckung *)

	(*Rüstsatz 206pol*)

	ST03_435_B67_4: sDigInVisu;		(*  Zuführung  frei zum Ablegen ISK SP Maschine Pos.1 *)
(*	ST03_425_B67_5: sDigInVisu;		(*  Zuführung  frei zum Ablegen ISK SP Maschine Pos.2 *)
	ST03_425_B67_6: sDigInVisu;		(*  Zuführung  frei zum Ablegen ISK SP Maschine Pos.3 *) *)
	ST03_435_B67_7: sDigInVisu;		(*  ISK anwesend am Vereinzler*)

	ST03_436_B68_1: sDigInVisu;		(*  Züführung  ISK auf Übergabeposition Roboter Palettierer 1*)
	ST03_436_B68_2: sDigInVisu;		(*  Züführung  ISK auf Übergabeposition Roboter Palettierer 2*)
	ST03_437_B68_4: sDigInVisu;		(*  Züführung  ISK auf Übergabeposition Roboter Palettierer*)
	ST03_437_Y68_5 : sValveVisu; 		(* Förderband  Zuführung Vereinzler AST/GST *)
	ST03_437_Y68_6 : sValveVisu; 		(* Förderband  Züführung Stopper AST/GST *)

(*Rüstsatz92pol*)

	ST03_444_B69_4: sDigInVisu;		(*  Zuführung  frei zum Ablegen ISK SP Maschine Pos.1 *)
	ST03_444_B69_7: sDigInVisu;		(*  ISK anwesend am Vereinzler*)

	ST03_445_B70_1: sDigInVisu;		(*  Züführung  ISK auf Übergabeposition Roboter Palettierer 1*)
	ST03_445_B70_2: sDigInVisu;		(*  Züführung  ISK auf Übergabeposition Roboter Palettierer 2*)
	ST03_446_B70_4: sDigInVisu;		(*  Züführung  ISK auf Übergabeposition Roboter Palettierer*)
	ST03_446_Y70_5 : sValveVisu; 		(* Förderband  Zuführung Vereinzler AST/GST *)
	ST03_446_Y70_6 : sValveVisu; 		(* Förderband  Züführung Stopper AST/GST *)


(*Rüstsatz124pol*)

	ST03_451_B69_4: sDigInVisu;		(*  Zuführung  frei zum Ablegen ISK SP Maschine Pos.1 *)
	ST03_451_B69_7: sDigInVisu;		(*  ISK anwesend am Vereinzler*)

	ST03_452_B70_1: sDigInVisu;		(*  Züführung  ISK auf Übergabeposition Roboter Palettierer 1*)
	ST03_452_B70_2: sDigInVisu;		(*  Züführung  ISK auf Übergabeposition Roboter Palettierer 2*)
	ST03_453_B70_4: sDigInVisu;		(*  Züführung  ISK auf Übergabeposition Roboter Palettierer*)
	ST03_453_Y70_5 : sValveVisu; 		(* Förderband  Zuführung Vereinzler AST/GST *)
	ST03_453_Y70_6 : sValveVisu; 		(* Förderband  Züführung Stopper AST/GST *)

(*Rüstsatz46pol*)

	ST03_461_B69_4: sDigInVisu;		(*  Zuführung  frei zum Ablegen ISK SP Maschine Pos.1 *)
	ST03_461_B69_7: sDigInVisu;		(*  ISK anwesend am Stopper*)

	ST03_462_B70_0: sDigInVisu;		(*   Förderband  ISK anwesend Wender*)
	ST03_462_B70_1: sDigInVisu;		(*  Züführung  ISK auf Übergabeposition Roboter Palettierer Lageerkennung 1*)
	ST03_462_B70_2: sDigInVisu;		(*  Züführung  ISK auf Übergabeposition Roboter Palettierer Lageerkennung 2*)
	ST03_463_B70_7: sDigInVisu;		(*  Züführung  ISK auf Übergabeposition Roboter Palettierer *)

	ST03_464_Y71_0 : sValveVisu; 		(* Förderband  Zuführung Vereinzelner Wendestation AST/GST *)
	ST03_464_Y71_1 : sValveVisu; 		(* Förderband  Zuführung Zylinder Vakuumdüsen AST/GST *)
	ST03_464_Y71_2 : sValveVisu; 		(* Förderband  Zuführung Wendestation Einlauf / Auslauf *)
	ST03_464_Y71_3 : sValveVisu; 		(* Förderband  Zuführung Vereinzler AST/GST *)
	ST03_464_Y71_4 : sValveVisu; 		(* Förderband  Zuführung Stopper AST/GST *)
	ST03_464_Y71_5 : sValveVisu; 		(* Förderband  Zuführung Vakuumdüsen EIN/AUS *)
	ST03_464_B71_6: sDigInVisu;		(* Förderband  Vakuum vorhanden *)
 	ST03_464_B71_7: sDigInVisu;		(*Förderband  Staustrecke mitte voll *)

(*Rüstsatz NOX 5+6 pol*)

	ST03_4x2_B69_0: sDigInVisu;		(*Zuführung frei zum Ablegen ISK SP Maschine *)
	ST03_4x2_B69_5: sDigInVisu;		(* ISK anwesend am Stopper *)

	ST03_4x3_B70_0: sDigInVisu;		(* ISK anwesend Übergabeposition Stopper*)
	ST03_4x3_B70_1: sDigInVisu;		(* ISK anwesend Übergabeposition*)

	ST03_4x3_Y70_5 : sValveVisu; 	(* Zuführung Vereinzler AST/GST *)
	ST03_4x3_Y70_6 : sValveVisu; 	(* Zuführung Stopper AST/GST *)
	ST03_4x3_Y70_7 : sValveVisu; 	(* Zuführung Stopper Übergabeposition AST/GST *)

(*Rüstsatz NOX 4 pol*)
	ST03_491_B69_0: sDigInVisu;		(*  Zuführung  frei zum Ablegen ISK SP Maschine*)
	ST03_491_B69_5: sDigInVisu;		(*  ISK anwesend am Stoper*)
	ST03_491_B69_7: sDigInVisu;		(*  ISK auf Abholposition Robi*)

	ST03_492_Y70_0 : sValveVisu; 		(* Förderband  Zuführung Vereinzler AST/GST *)
	ST03_492_Y70_1 : sValveVisu; 		(* Förderband  Züführung Stopper AST/GST *)

(*Rüstsatz 88 pol*)
	ST03_501_B69_0: sDigInVisu;		(*  Zuführung  frei zum Ablegen ISK SP Maschine*)

	ST03_501_B69_5: sDigInVisu;		(*  ISK anwesend am Vereinzler*)
	ST03_501_B69_6: sDigInVisu;		(*  ISK anwesend am Stoper*)
	ST03_501_B69_7: sDigInVisu;		(*  ISK auf Abholposition Robi*)

	ST03_502_B70_0: sDigInVisu;		(*  ISK Lageerkennung*)
	ST03_502_Y70_1 : sValveVisu; 		(* Förderband  Zuführung Vereinzler AST/GST *)
	ST03_502_Y70_2 : sValveVisu; 		(* Förderband  Züführung Stopper AST/GST *)

(*Rüstsatz 7 pol*)
	ST03_512_XG1:    sDigInVisu;			(*  ISK in Rinne*)
	ST03_514_B71_7: sDigInVisu;		(*  Führungsschiene frei zum schwenken*)

	ST03_513_B70_4: sDigInVisu;		(*  ISK anwesend am Stoper*)
	ST03_513_B70_7: sDigInVisu;		(*  ISK auf Übergabeposition 1*)

	ST03_514_B71_2: sDigInVisu;		(*  ISK auf Übergabeposition 2*)
	ST03_514_B71_5: sDigInVisu;		(*  ISK auf Übergabeposition 3*)
	ST03_514_B71_6: sDigInVisu;		(*  ISK auf Übergabeposition 4*)

	ST03_515_Y72_0 : sValveVisu; 		(* SK Klemmen in Rinne AST/GST *)
	ST03_515_Y72_1 : sValveVisu; 		(* Rinne schwenkern AST/GST *)
	ST03_515_Y72_2 : sValveVisu; 		(* Führungsschiene  Zuführung Vereinzler AST/GST *)
	ST03_515_Y72_3 : sValveVisu; 		(* Führungsschiene  Zuführung Stopper AST/GST *)
	ST03_515_Y72_4 : sValveVisu; 		(* Übergabeposition Stopper 1  AST/GST *)
	ST03_515_Y72_5 : sValveVisu; 		(* Übergabeposition Stopper 2  AST/GST *)
	ST03_515_Y72_6 : sValveVisu; 		(* Übergabeposition Stopper 3  AST/GST *)

(*Rüstsatz 88 pol AMG*)
	ST03_521_B69_0: sDigInVisu;			(*Zuführung  frei zum Ablegen ISK SP Maschine*)

	ST03_521_B69_6: sDigInVisu;			(*ISK anwesend am Stopper*)
	ST03_521_B69_7: sDigInVisu;			(*ISK Lageerkennung links*)

	ST03_522_B70_0: sDigInVisu;			(*ISK Lageerkennung rechts*)
	ST03_522_Y70_1 : sValveVisu; 		(*Zuführung Vereinzler AST/GST *)
	ST03_522_Y70_2 : sValveVisu; 		(*Züführung Stopper AST/GST*)

(*Rüstsatz 120 pol *)
	ST03_531_B69_0: sDigInVisu;			(*Zuführung  frei zum Ablegen ISK SP Maschine*)

	ST03_531_B69_6: sDigInVisu;			(*ISK anwesend am Stopper*)
	ST03_531_B69_7: sDigInVisu;			(*ISK rechts Lageerkennung*)

	ST03_532_B70_0: sDigInVisu;			(*ISK links Lageerkennung *)
	ST03_532_Y70_1 : sValveVisu; 		(*Zuführung Vereinzler AST/GST *)
	ST03_532_Y70_2 : sValveVisu; 		(*Züführung Stopper AST/GST*)

(*Rüstsatz 21 pol *)
	ST03_536_B69_0: sDigInVisu;			(*Zuführung  frei zum Ablegen ISK SP Maschine*)

	ST03_536_B69_6: sDigInVisu;			(*ISK anwesend am Stopper*)
	ST03_536_B69_7: sDigInVisu;			(*ISK anwesend an Abholposition*)

	ST03_537_B70_0: sDigInVisu;			(*ISK Lageerkennung *)
	ST03_537_Y70_1 : sValveVisu; 		(*Zuführung Vereinzler AST/GST *)
	ST03_537_Y70_2 : sValveVisu; 		(*Züführung Stopper AST/GST*)

(*Rüstsatz 191 pol *)
	ST03_541_B69_0: sDigInVisu;			(*Zuführung  frei zum Ablegen ISK SP Maschine*)

	ST03_541_B69_6: sDigInVisu;			(*ISK anwesend am Stopper*)
	ST03_541_B69_7: sDigInVisu;			(*ISK rechts Lageerkennung*)

	ST03_542_B70_0: sDigInVisu;			(*ISK links Lageerkennung*)
	ST03_542_Y70_1 : sValveVisu; 		(*Zuführung Vereinzler AST/GST *)
	ST03_542_Y70_2 : sValveVisu; 		(*Züführung Stopper AST/GST*)

(*Rüstsatz  72pol *)
	ST03_546_B69_0: sDigInVisu;			(*Zuführung  frei zum Ablegen ISK SP Maschine*)

	ST03_546_B69_6: sDigInVisu;			(*ISK anwesend am Stopper*)
	ST03_546_B69_7: sDigInVisu;			(*ISK rechts Lageerkennung*)

	ST03_547_B70_0: sDigInVisu;			(*ISK links Lageerkennung*)
	ST03_547_Y70_1 : sValveVisu; 		(*Zuführung Vereinzler AST/GST *)
	ST03_547_Y70_2 : sValveVisu; 		(*Züführung Stopper AST/GST*)

(*Rüstsatz 48 pol *)
	ST03_551_B69_0: sDigInVisu;			(*Zuführung  frei zum Ablegen ISK SP Maschine*)

	ST03_551_B69_6: sDigInVisu;			(*ISK anwesend am Stopper*)
	ST03_551_B69_7: sDigInVisu;			(*ISK rechts Lageerkennung*)

	ST03_552_B70_0: sDigInVisu;		(*ISK links Lageerkennung*)
	ST03_552_Y70_1 : sValveVisu; 		(*Zuführung Vereinzler AST/GST *)
	ST03_552_Y70_2 : sValveVisu; 		(*Züführung Stopper AST/GST*)

(*Rüstsatz 268 pol *)
	ST03_556_B69_0: sDigInVisu;		(*Zuführung  frei zum Ablegen ISK SP Maschine*)

	ST03_556_B69_5: sDigInVisu;		(* Führungsschiene Überwachung Staustrecke*)
	ST03_556_B69_6: sDigInVisu;		(*ISK anwesend am Stopper*)
	ST03_556_B69_7: sDigInVisu;		(*ISK anwesend an Abholposition*)

	ST03_557_Y70_1 : sValveVisu; 		(*Zuführung Vereinzler AST/GST *)
	ST03_557_Y70_2 : sValveVisu; 		(*Züführung Stopper AST/GST*)

(*Rüstsatz 268 pol Rasterplatte======================================================================================*)
	ST03_562_B69_0: sDigInVisu;		(*Zuführung 1 frei zum schwenken*)
	ST03_562_B69_6: sDigInVisu;		(*Zuführung 1 ISK anwesend am Stopper*)
	ST03_562_B67_7: sDigInVisu;		(*Zuführung 1 ISK auf Übergabepos. Robi*)

	ST03_563_B70_0: sDigInVisu;		(*Zuführung 2 frei zum schwenken*)
	ST03_563_B70_6: sDigInVisu;		(*Zuführung 2 ISK anwesend am Stopper*)
	ST03_563_B70_7: sDigInVisu;		(*Zuführung 2 ISK auf Übergabepos. Robi*)

	ST03_564_Y71_0: sValveVisu; 		(*Zuführung 1 Vereinzler AST/GST *)
	ST03_564_Y71_1: sValveVisu; 		(*Zuführung 1 Stopper AST/GST *)
	ST03_564_Y71_2: sValveVisu; 		(*Zuführung 2 Vereinzler AST/GST *)
	ST03_564_Y71_3: sValveVisu; 		(*Zuführung 2 Stopper AST/GST *)
	ST03_564_Y71_4: sValveVisu; 		(* ISK Klemmer AST/GST *)
	ST03_564_Y71_5: sValveVisu; 		(* Rinne schwenkern AST/GST *)

	ST03_565_B72_0: sDigInVisu;		(* ISK 1 in Klemmer*)
	ST03_565_B72_1: sDigInVisu;		(* ISK 2 in Klemmer*)

(*Rüstsatz 33 pol Rasterplatte======================================================================================*)
	ST03_571_B69_0	: sDigInVisu;		(* Zuführung  Pos 1 frei zum Ablegen ISK SP Maschine*)
	ST03_571_B69_1	: sDigInVisu;		(* Zuführung  Pos 2 frei zum Ablegen ISK SP Maschine*)

	ST03_571_B69_6	: sDigInVisu;		(* ISK anwesend am Stopper*)
	ST03_571_B69_7	: sDigInVisu;		(* ISK anwesend an Abholposition*)

	ST03_572_Y70_0	: sValveVisu; 		(* Zuführung Vereinzler AST/GST *)
	ST03_572_Y70_1	: sValveVisu; 		(* Züführung Stopper AST/GST *)

(*---------------------------------------------------------------------------
  Station08
  ---------------------------------------------------------------------------*)


	ST08_170_Q2 : sDigInVisu; (* Bandstrecken Station 8 Motorschutz i.O. *)
	ST08_170_M : sDigInVisu; (* Bandstrecken Station 8 Thermokontakt i.O. *)

	ST08_400_B50_0 : sDigInVisu; (* Traystapel vor Vereinzeler Einlaufband hinten *)
	ST08_401_B50_5 : sDigInVisu; (* Traystapel vor Vereinzeler Einlaufband mitte *)
	ST08_402_B51_2 : sDigInVisu; (* Traystapel vor Vereinzeler Einlaufband vorne *)
	ST08_402_B51_4 : sDigInVisu; (* Luftzone 1 *)
	ST08_402_B51_5 : sDigInVisu; (* Luftzone 2 *)
	ST08_404_B52_2 : sDigInVisu; (* Traystapel in Ablageposition Isokörper *)
	ST08_404_B52_3 : sDigInVisu; (* Traystapel richtig eingelegt Isokörper *)
	ST08_406_B54_0 : sDigInVisu; (* Tray in Zwischenp. Entnahme Isokörper (Bandende) *)
	ST08_406_B54_3 : sDigInVisu; (* Tray in Ausheber. Entnahme Isokörper (Bandende) *)
	ST08_406_B54_6 : sDigInVisu; (* Tray aus Entnahme ausgelaufen (Bandende) *)
	ST08_407_B55_1 : sDigInVisu; (* Tray aus entnahme ausgelaufen STN8 *)
	ST08_407_B55_4 : sDigInVisu; (* Tray in Aufstapelposition eingelaufen STN8 *)
	ST08_409_B55_5 : sDigInVisu; (* Auslaufrollenbahn voll STN8 *)

	ST08_412_B58_4: sDigInVisu;		(*  Rüstsatz Förderband frei zum Ablegen ISK von SP Maschine Position 1 *)
	ST08_412_B58_5: sDigInVisu;		(*  Rüstsatz Förderband frei zum Ablegen ISK von SP Maschine Position 2 *)
	ST08_412_B58_6: sDigInVisu;		(*  Rüstsatz Förderband frei zum Ablegen ISK von SP Maschine Position 3 *)
	ST08_412_B58_5_35pol: sDigInVisu;		(*  Lageerkennung links *)
	ST08_412_B58_6_35pol: sDigInVisu;		(*  Lageerkennung rechts *)
	ST08_412_B58_7: sDigInVisu;		(*  Rüstsatz Förderband ISK anwesend zum Vereinzeln *)
	ST08_412_B59_0: sDigInVisu;		(*  Rüstsatz Förderband ISK auf Übergabeposition Roboter Verpackung *)

	ST08_169_K1 : sDigOutInVisu; (* Bandantrieb 1 Einlauf Trays Ein *)
	ST08_169_K2 : sDigOutInVisu; (* Bandantrieb 4 Auslauf leere Trays Ein *)
	ST08_170_K1 : sDigOutInVisu; (* Bandantrieb 2 Hubquereinheit Trays Ein *)
	ST08_170_K2 : sDigOutInVisu; (* Bandantrieb 3 Hubquereinheit Trays Ein *)

	ST08_400_Y50_0 : sValveVisu; (* Stopper Traystapel Einlaufb. hinten links + rechts AST *)
	ST08_400_Y50_2 : sValveVisu; (* Stopper Traystapel Einlaufb. mitte links + rechts AST *)
	ST08_402_Y50_4 : sValveVisu; (* Stopper Traystapel Einlaufb. vorne links + rechts AST *)
	ST08_403_Y50_6 : sValveVisu; (* Vakuum 1 Einlauf STN8 AST *)
	ST08_403_Y50_7 : sValveVisu; (* Vakuum 2 Einlauf STN8 AST *)
	ST08_405_Y51_0 : sValveVisu; (* Hubtüre 2 Einlauf Isokörper STN8 AST *)
	ST08_404_Y51_6 : sValveVisu; (* Stopper Traystapel Isokörper AST *)
	ST08_406_Y51_2 : sValveVisu; (* Hubtüre 3 STN8 AST *)
	ST08_407_Y51_4 : sValveVisu; (* Hubtüre 4 Auslauf STN8 AST *)
	ST08_404_Y52_0 : sValveVisu; (* Hub Bandstrecke AST *)
	ST08_406_Y52_3 : sValveVisu; (* Ausheber Trays Entnahmepos. Isok. STN8 GST *)
	ST08_401_Y52_4 : sValveVisu; (* Traystapel schieben hinte AST *)
	ST08_400_Y52_5 : sValveVisu; (* Stopper links + rechts Traystapel Auslaufband einfahren *)
	ST08_402_Y52_6 : sValveVisu; (* Traystapel schieben mitte AST *)
	ST08_402_Y52_7 : sValveVisu; (* Traystapel schieben vorne AST *)
	ST08_404_Y53_0 : sValveVisu; (* Abstapelzylinder 1 Isokörper AST *)
	ST08_404_Y53_2 : sValveVisu; (* Abstapelzylinder 2 Isokörper AST *)
	ST08_405_Y53_4 : sValveVisu; (* Rückhaltezylinder li+re Traystapel Isokörper AST *)
	ST08_408_Y54_0 : sValveVisu; (* Rückhaltezylinder li.+re. Auslauf STN8 AST *)
	ST08_408_Y54_2 : sValveVisu; (* Abstapelzylinder 1 STN8 AST *)
	ST08_408_Y54_4 : sValveVisu; (* Abstapelzylinder 2 STN8 AST *)

	ST08_412_Y55_0 : sValveVisu; (* Rüstsatz Förderband Vereinzelner *)
	ST08_412_Y55_2 : sValveVisu; (* Rüstsatz Förderband Stopper *)

	ST08_180_M1 		: sDigInVisu; (* Abstapeln *)
	ST08_185_M1 		: sDigInVisu; (* Aufstapeln *)
	ST08_190_M1 		: sDigInVisu; (* Tray ausheben *)

END_STRUCT
END_TYPE

(* Data type in sStation *)
TYPE PartState :
(
	PART_NO			:= 0, (*no Part available*)
	PART_OK			:= 1, (*Part processed with OK-Result*)
	PART_NOK		:= 2, (*Part processed with NOK-Result*)
	PART_NEW		:= 4,  (*new Part (picked up from Feeder, and not yet processed) *)
	PART_CAM		:= 5	(*Part muss zur Kamera*)
);
END_TYPE

(* Data type in sStation *)
TYPE SFCCurrent :
STRUCT
	SFCCurrentPOU		: STRING:=	'-';
	SFCCurrentStep		: STRING;
	SFCTime			: DINT;
	b_activ				: BOOL;
END_STRUCT
END_TYPE

(* Data type in System/Error_and_Message *)
TYPE eMsgDataLineType :
	(
	MsgDataTypeNone			:=	0,
	MsgDataTypeBool			:=	1,
	MsgDataTypeDint			:=	2,
	MsgDataTypeReal			:=	3,
	MsgDataTypeString		:=	4
	);
END_TYPE

(* Data type in System/Error_and_Message *)
TYPE ErrorStruct :
STRUCT
	No							: DINT;
	DateTime					: DT;
	Text						: STRING(255);
	Typ							: DINT; (* 0=FatalError , 1=Warning, 2=OperatorInfo *)
	Station						: DINT;
	Prio						: DINT; (*1=heighest, .. , 4=lowest*)
	QuitAddr					: DWORD;
	LineColor					: DINT;
(*	Instance					: STRING;*)
END_STRUCT
END_TYPE

(* Data type in System/Error_and_Message *)
TYPE sErrorHandlerVisu :
STRUCT
	Error								:	ARRAY[0..NO_OF_ERRORS] OF ErrorStruct;
	ScrollBarShow				:	BOOL;
	ScrollBarMax				:	DINT;
	ScrollBarPosition		:	DINT;
END_STRUCT
END_TYPE

(* Data type in System/Error_and_Message *)
TYPE sMessageLine :
STRUCT
	Visible				: BOOL;
	Editable			: BOOL;
	Text		    	: STRING(80);
	MsgTypeEnum		: eMsgDataLineType; (*BOOL, DINT, REAL, STRING *)
	MsgType				: STRING; (*BOOL, DINT, REAL, STRING *)
	MsgBool	  	  : BOOL;
	MsgInt		    : DINT;
	MsgReal			  : REAL;
	MsgString			: STRING(40);
END_STRUCT
END_TYPE

(* Data type in System/Error_and_Message *)
TYPE sMessageText :
STRUCT
	ShowMessage				: BOOL;
	ID							: STRING(20);
	Name						: STRING(30);
	Text						: STRING(160);
	Color						: DINT; (*from STRUCT Colors*)
	DateTime					: DT;
	Station						: DINT;
	Button1						: sButtonVisu;
	Button2						: sButtonVisu;
END_STRUCT
END_TYPE

(* Data type in System/Error_and_Message *)
TYPE sMessageVisu :
STRUCT
	ShowMessage			: BOOL;
	ID						: STRING(20);
	Name					: STRING(30);
	Text					: STRING(255);
	Color					: DINT; (*from STRUCT Colors*)
	DateTime				: DT;
	Station					: DINT;
	Button1					: sButtonVisu;
	Button2					: sButtonVisu;
	MessageLine			: ARRAY [1..10] OF sMessageLine;

	BtnHide					: sButtonVisu;
	BtnShow					: sButtonVisu;
	TextMinimized			: STRING(60);
END_STRUCT
END_TYPE

(* Data type in System/GlobalStates *)
TYPE StateMode :
(
(* different modes of the Mode-Dispatcher
   verschiedene Betriebsarten des Betriebsartenbausteines *)
	MODE_NON					:= 0,		(*MODE_NON*)
	MODE_MANUAL				:= 10,		(*MODE_MANUAL*)
	MODE_STEP					:= 20,		(*MODE_STEP*)
	MODE_STEP_RUN				:= 21,		(*MODE_STEP_RUN*)
	MODE_STEP_STOP			:= 22,		(*MODE_STEP_STOP*)
	MODE_AUTO					:= 30,		(*MODE_AUTO*)
	MODE_AUTO_RUN				:= 31,		(*MODE_AUTO_RUN*)
	MODE_AUTO_STOP 			:= 32,		(*MODE_AUTO_STOP*)
	MODE_HOME_POS_RUN		:= 40,		(*MODE_HOME_POS_RUN*)
	MODE_SPECIAL				:= 50 		(*MODE_SPECIAL*)
);
END_TYPE

(* Data type in System/GlobalStates *)
TYPE StateObject :
	(
	STATE_ERROR			:= -1,  		 (*STATE_ERROR Objekt meldet Fehler *)
	STATE_TIMEOUT  		:= -2,	 	  (*STATE_TIMEOUT Objekt meldet Fehler *)
	STATE_UNDEFINED		:= 0,		(*STATE_UNDEFINED Das Objekt befindet sich in einem undefinierten Zustand *)
	STATE_OK			:= 1,		(*STATE_OK Die letzte Aktion wurde erfolgreich durchgeführt *)
	STATE_RUN			:= 2,		(*STATE_RUN Die Aktion wird gerade durchgeführt *)
	STATE_WAIT			:= 3,		(*STATE_WAIT Bereit (für neue Aktion) *)
	STATE_STOPPED		:= 4,		(*STATE_STOPPED Objekt gesperrt(durch externes Enable) *)
	STATE_RESETS		:= 5,		(*STATE_RESETS Objekt wird zurückgesetzt *)
	STATE_IGNORED		:= 6 		(*STATE_IGNORED Alle Stati und Meldungen werden ignoriert *)
	);
END_TYPE

(* Data type in System/GlobalStates *)
TYPE StateResult :
(
	RESULT_NON 			:=	0,  (* No Result from sequence *)
	RESULT_OK			:=	1,	(* End of Sequence with OK *)
	RESULT_NOK			:=	2,	(* End of Sequence with NOT OK *)
	RESULT_REW			:=	3 	(* End of Sequence with REWORK *)

);
END_TYPE

(* Data type in System/LanguageHandler *)
TYPE enum_Lng :
(
	DE 			:=	0,
	EN			:=	1,
	CZ			:=	2

);
END_TYPE

(* Data type in System/LoginDialog *)
TYPE sNumericKeypad :
STRUCT
		Visible					:	BOOL;
		Enable					:	BOOL;

		btn_Key1						:	sButtonVisu;
		btn_Key2						:	sButtonVisu;
		btn_Key3						:	sButtonVisu;
		btn_Key4						:	sButtonVisu;
		btn_Key5						:	sButtonVisu;
		btn_Key6						:	sButtonVisu;
		btn_Key7						:	sButtonVisu;
		btn_Key8						:	sButtonVisu;
		btn_Key9						:	sButtonVisu;
		btn_Key0						:	sButtonVisu;
		btn_KeyDot					:	sButtonVisu;

		btn_KeyBack					:	sButtonVisu;
		btn_KeyEsc					:	sButtonVisu;
		btn_KeyClear				:	sButtonVisu;
		btn_KeyOK 					:	sButtonVisu;
		btn_KeyVorzeichen		:	sButtonVisu;


		InputString			:	STRING;

END_STRUCT
END_TYPE

(* Data type in System/LoginDialog *)
TYPE sUserData :
STRUCT
	UserName						: STRING;
	UserPassword					: STRING;
	UserLevel						: INT;
	UserCanChangeOwnPassword		: BOOL;
END_STRUCT
END_TYPE

(* Data type in System/LoginDialog *)
TYPE sVisuLoginDialog :
STRUCT

	LoginKeyPad			: sNumericKeypad;
	btn_Login			: sButtonVisu;
	btn_LogOut			: sButtonVisu;
	btn_ChangeUserData	: sButtonVisu;
	btn_ChangePassword	: sButtonVisu;

	ShowEditFields		: BOOL;
	UserListIndex		: INT;

	UserEdit			: sUserData;

END_STRUCT
END_TYPE

(* Data type in System/MachineParameterHandler *)
TYPE sMPHandler :
STRUCT

	FileListExport				: ARRAY[1..20] OF STRING(80);
	FileListLocal					: ARRAY[1..20] OF STRING(80);

	FileNameSelected			: STRING(80);
	FileNameSaveAs			: STRING(80);

	FileIndex					: DINT;
	FileFilter						: STRING(80);

	FileListUpdate				: BOOL;

	BtnImport					: sButtonVisu;
	BtnExport					: sButtonVisu;

	MessageString				: STRING;

END_STRUCT
END_TYPE

(* Data type in System/MP_ShiftHandler *)
TYPE sMP_ShiftData :
STRUCT
	ShiftName			: STRING;
	ShiftIndex		: DINT;
	ShiftActive		: BOOL;
	TimeStart			: Timestruct;
	TimeEnd				: Timestruct;

END_STRUCT
END_TYPE

(* Data type in System/MP_ShiftHandler *)
TYPE sMP_ShiftHandler :
STRUCT
	ActiveShift	:	sMP_ShiftData;
	Shift				: ARRAY[1..3] OF sMP_ShiftData;
END_STRUCT
END_TYPE

(* Data type in System/SystemSettings *)
TYPE eTargetSystem :
	(
	TARGETSYSTEM_CE					:=  1,   (* TaragetSystem with Winwows CE *)
	TARGETSYSTEM_XPP				:=  2,   (* TaragetSystem with Winwows XP Pro SP 3 *)
	TARGETSYSTEM_LOCAL_C		:=  3,   (* TaragetSystem on Developmant System - Path Mapped to Drive C *)
	TARGETSYSTEM_LOCAL_D		:=  4    (* TaragetSystem on Developmant System - Path Mapped to Drive D *)
	);
END_TYPE

(* Data type in System/TypeDataHandler *)
TYPE sTDHandler :
STRUCT
	TypeDataValid			: BOOL;

	FileList					: ARRAY[1..NO_OF_FILES] OF STRING(80);
	FileNameSelected		: STRING(80);
	FileNameSaveAs		: STRING(80);

	FileListUpdate			: BOOL;
	FileIndex				: DINT:=1;
	FileFilter					: STRING(80);

	BtnLoad				: sButtonVisu;
	BtnSave				: sButtonVisu;
	BtnSaveAs				: sButtonVisu;
	BtnActivate				: sButtonVisu;
	BtnClose				: sButtonVisu;
	BtnDelete				: sButtonVisu;
	BtnNew					: SButtonVisu;

END_STRUCT
END_TYPE

(* Data type in System/VisuInterface *)
TYPE sButtonVisu :
STRUCT
		Visible				: BOOL;
		Enable				: BOOL;
		Pressed				: BOOL;
		Text				: STRING;
		TextColor			: DINT;
		BackgroundColor	: DINT ;
		Tasten				: BOOL;
END_STRUCT
END_TYPE

(* Data type in System/VisuInterface *)
TYPE sButtonVisu_Tree :
STRUCT
	unsichtbar				: BOOL;
	deaktivieren				: BOOL;
	tasten					: BOOL;
	Textfarbe				: DINT;
	innenFarbe				: DINT;
	Text					: STRING(50);
	Zoom					: STRING(50);
END_STRUCT
END_TYPE

(* Data type in System/VisuInterface *)
TYPE sButtonVisuBmp :
STRUCT
	unsichtbar			: BOOL;
	deaktivieren		: BOOL;
	tasten				: BOOL;
	Text				: STRING(30);
	Textfarbe			: DINT;
	innenFarbe			: DINT;
	BmpPath				: STRING(255);
END_STRUCT
END_TYPE

(* Data type in System/VisuInterface *)
TYPE sColorCode :
STRUCT
	black				:    DINT  :=  16#000000;
	maroon   			:    DINT  :=  16#000080;
	green  				:    DINT  :=  16#008000;
	olive    				:    DINT  :=  16#008080;
	navy    				:    DINT  :=  16#800000;
	purple    			:    DINT  :=  16#800080;
	teal    				:    DINT  :=  16#808000;
	grey    				:    DINT  :=  16#808080;
	silver    			:    DINT  :=  16#C0C0C0;
	red    				:    DINT  :=  16#0000FF;
	lime    				:    DINT  :=  16#00FF00;
	yellow    			:    DINT  :=  16#00FFFF;
	blue    				:    DINT  :=  16#FF0000;
	fuchsia    			:    DINT  :=  16#FF00FF;
	aqua    			:    DINT  :=  16#FFFF00;
	white    			:    DINT  :=  16#FFFFFF;
	aliceblue    		:    DINT  :=  16#FFF8F0;
	antiquewhite   	:    DINT  :=  16#D7EBFA;
	aquamarine    :    DINT  :=  16#D4FF7F;
	azure    			:    DINT  :=  16#FFFFF0;
	beige    			:    DINT  :=  16#DCF5F5;
	blueviolet    	:    DINT  :=  16#E22B8A;
	brown    			:    DINT  :=  16#2A2AA5;
	burlywood    	:    DINT  :=  16#87B8DE;
	cadetblue    :    DINT  :=  16#A09E5F;
	chartreuse    :    DINT  :=  16#00FF7F;
	chocolate    :    DINT  :=  16#1E69D2;
	coral    :    DINT  :=  16#507FFF;
	cornflowerblue    :    DINT  :=  16#ED9564;
	cornsilk    :    DINT  :=  16#DCF8FF;
	crimson    :    DINT  :=  16#3C14DC;
	darkblue    :    DINT  :=  16#8B0000;
	darkcyan    :    DINT  :=  16#8B8B00;
	darkgoldenrod    :    DINT  :=  16#0B86B8;
	darkgrey    :    DINT  :=  16#A9A9A9;
	darkgreen    :    DINT  :=  16#006400;
	darkkhaki    :    DINT  :=  16#6BB7BD;
	darkmagenta    :    DINT  :=  16#8B008B;
	darkolivegreen    :    DINT  :=  16#2F6B55;
	darkorange    :    DINT  :=  16#008CFF;
	darkorchid    :    DINT  :=  16#CC3299;
	darkred    :    DINT  :=  16#00008B;
	darksalmon    :    DINT  :=  16#7A96E9;
	darkseagreen    :    DINT  :=  16#8FBC8F;
	darkslateblue    :    DINT  :=  16#8B3D48;
	darkslategrey    :    DINT  :=  16#4F4F2F;
	darkturquoise    :    DINT  :=  16#D1CE00;
	darkviolet    :    DINT  :=  16#D30094;
	deeppink    :    DINT  :=  16#9314FF;
	deepskyblue    :    DINT  :=  16#FFBF00;
	dimgrey    :    DINT  :=  16#696969;
	dodgerblue    :    DINT  :=  16#FF901E;
	firebrick    :    DINT  :=  16#2222B2;
	floralwhite    :    DINT  :=  16#F0FAFF;
	forestgreen    :    DINT  :=  16#228B22;
	gainsboro    :    DINT  :=  16#DCDCDC;
	ghostwhite    :    DINT  :=  16#FFF8F8;
	gold    :    DINT  :=  16#00D7FF;
	goldenrod    :    DINT  :=  16#20A5DA;
	greenyellow    :    DINT  :=  16#2FFFAD;
	honeydew    :    DINT  :=  16#F0FFF0;
	hotpink    :    DINT  :=  16#B469FF;
	indianred    :    DINT  :=  16#5C5CCD;
	indigo    :    DINT  :=  16#82004B;
	ivory    :    DINT  :=  16#F0FFFF;
	khaki    :    DINT  :=  16#8CE6F0;
	lavender    :    DINT  :=  16#FAE6E6;
	lavenderblush    :    DINT  :=  16#F5F0FF;
	lawngreen    :    DINT  :=  16#00FC7C;
	lemonchiffon    :    DINT  :=  16#CDFAFF;
	lightblue    :    DINT  :=  16#E6D8AD;
	lightcoral    :    DINT  :=  16#8080F0;
	lightcyan    :    DINT  :=  16#FFFFE0;
	lightgoldenrodyellow    :    DINT  :=  16#D2FAFA;
	lightgreen    :    DINT  :=  16#90EE90;
	lightgrey    :    DINT  :=  16#D3D3D3;
	lightpink    :    DINT  :=  16#C1B6FF;
	lightsalmon    :    DINT  :=  16#7AA0FF;
	lightseagreen    :    DINT  :=  16#AAB220;
	lightskyblue    :    DINT  :=  16#FACE87;
	lightslategrey    :    DINT  :=  16#998877;
	lightsteelblue    :    DINT  :=  16#DEC4B0;
	lightyellow    :    DINT  :=  16#E0FFFF;
	limegreen    :    DINT  :=  16#32CD32;
	linen    :    DINT  :=  16#E6F0FA;
	mediumaquamarine    :    DINT  :=  16#AACD66;
	mediumblue    :    DINT  :=  16#CD0000;
	mediumorchid    :    DINT  :=  16#D355BA;
	mediumpurple    :    DINT  :=  16#D7093;
	mediumseagreen    :    DINT  :=  16#71B33C;
	mediumslateblue    :    DINT  :=  16#EE687B;
	mediumspringgreen    :    DINT  :=  16#9AFA00;
	mediumturquoise    :    DINT  :=  16#CCD148;
	mediumvioletred    :    DINT  :=  16#8515C7;
	midnightblue    :    DINT  :=  16#701919;
	mintcream    :    DINT  :=  16#FAFFF5;
	mistyrose    :    DINT  :=  16#E1E4FF;
	moccasin    :    DINT  :=  16#B5E4FF;
	navajowhite    :    DINT  :=  16#ADDEFF;
	oldlace    :    DINT  :=  16#E6F5FD;
	olivedrab    :    DINT  :=  16#238E6B;
	orange    :    DINT  :=  16#00A5FF;
	orangered    :    DINT  :=  16#0045FF;
	orchid    :    DINT  :=  16#D670DA;
	palegoldenrod    :    DINT  :=  16#AAE8EE;
	palegreen    :    DINT  :=  16#98FB98;
	paleturquoise    :    DINT  :=  16#EEEEAF;
	palevioletred    :    DINT  :=  16#9370DB;
	papayawhip    :    DINT  :=  16#D5EFFF;
	peachpuff    :    DINT  :=  16#B9DAFF;
	peru    :    DINT  :=  16#3F85CD;
	pink    :    DINT  :=  16#CBC0FF;
	plum    :    DINT  :=  16#DDA0DD;
	powderblue    :    DINT  :=  16#E6E0B0;
	rosybrown    :    DINT  :=  16#8F8FBC;
	royalblue    :    DINT  :=  16#E16941;
	saddlebrown    :    DINT  :=  16#13458B;
	salmon    :    DINT  :=  16#7280FA;
	sandybrown    :    DINT  :=  16#60A4F4;
	seagreen    :    DINT  :=  16#578B2E;
	seashell    :    DINT  :=  16#EEF5FF;
	sienna    :    DINT  :=  16#2D52A0;
	skyblue    :    DINT  :=  16#EBCE87;
	slateblue    :    DINT  :=  16#CD5A6A;
	slategrey    :    DINT  :=  16#908070;
	snow    :    DINT  :=  16#FAFAFF;
	springgreen    :    DINT  :=  16#7FFF00;
	steelblue    :    DINT  :=  16#B48246;
	thistle    :    DINT  :=  16#D8BFD8;
	tomato    :    DINT  :=  16#4763FF;
	turquoise    :    DINT  :=  16#D0E040;
	violet    :    DINT  :=  16#EE82EE;
	wheat    :    DINT  :=  16#B3DEF5;
	whitesmoke    :    DINT  :=  16#F5F5F5;
	yellowgreen    :    DINT  :=  16#32CD9A;
 	control    :    DINT  :=  16#D3D3D3;
(*	control    :    DINT  :=  16#D8E9EC;*)



END_STRUCT
END_TYPE

(* Data type in System/VisuInterface *)
TYPE sModeSelectInit :
STRUCT
	(* Structure for initialising the object *)
	(* Initialisierungsstruktur des Objektes *)

	InstName							:	STRING(16);		(* Instanzname of the object *)
																				(* Name der Instanz *)
	EnableQuickAutoStart 	: BOOL;     		(* If TRUE, then show AutoStartButton in MODE_AUTO always:
                                    			          if HomePosition=FALSE then change first in MODE=MODE_HOME_POS_RUN *) 
	RemoteAutoStopToManual: BOOL;     		(* If TRUE, then the mode change to MODE=MODE_MANUAL
                                   				          if FALSE then change to MODE=MODE_AUTO_STOP *) 

	HideManualButton			:	BOOL;     		(* If TRUE, then hide ManualMode-Button (then ManuelMode is not used)*)
	HideNextStepButton		:	BOOL;     		(* If TRUE, then hide StepMode-Button (then StepMode is not used)*)
END_STRUCT
END_TYPE

(* Data type in System/VisuInterface *)
TYPE sModeSelectVisu :
STRUCT

	BtnManual		: sButtonVisu;
	BtnStep			: sButtonVisu;
	BtnStepCycle: sButtonVisu;
	BtnAuto			: sButtonVisu;
	BtnAutoStart: sButtonVisu;
	BtnAutoStop	: sButtonVisu;
	BtnRunEmpty	: sButtonVisu;
	BtnHomeRun	: sButtonVisu;
	BtnSpecial	: sButtonVisu;
	BtnSpecStep	: sButtonVisu;
	BtnReset		: sButtonVisu;

	ManualOn					:	BOOL;		(*manual-mode is activ*)
	StepOn						:	BOOL;		(*step-mode is activ*)
	AutoOn						:	BOOL;		(*auto-mode is activ*)
	AutoStartOn				:	BOOL;		(*automatic is running*)
	AutoStopOn				:	BOOL;		(*automaticv running in last cycle*)
	RunEmptyOn				:	BOOL;		(*machine is running empty*)
	HomePosRunOn			:	BOOL;		(*home-position-run is activ*)
	SpecialOn					:	BOOL;		(*special-mode is activ*)

	BasicManualMode		:	BOOL;		(*the basic-mode 'manual' is activ*)
	BasicAutoMode			:	BOOL; 	(*the basic-mode 'automatic' is activ*)
															(*auto, autostart, autostop, step, homeposrun*)
	HomePositionOk		:	BOOL;		(* home position *)
	HomePositionInfoNo: DINT;		(* missing to home position *)
	DisableString			: STRING(50);	(* string shows missing signal *)
															(* string zeigt fehlende Bedingung an *)
	State							:	DINT;		(*status-messages from mode-dispatcher*)
END_STRUCT
END_TYPE

(* Data type in zLibrary/AnaIn *)
TYPE enum_Drehrichtung :
	(
	RUECKWAERTS := -1,
	STEHT := 0,
	VORWAERTS := 1
	);
END_TYPE

(* Data type in zLibrary/AnaIn *)
TYPE sAnaInInit :
STRUCT
	InstName				:STRING(20);	(* Name of instance  *)
	Description				:STRING(32);	(* Description  *)
	BitInName				:STRING(25);	(* Name of bit input *)
	ScalingSensorValueMin	:INT;			(* min Scaling Value from Sensor *)
	ScalingSensorValueMax	:INT;			(* max Scaling Value from Sensor *)
	ScalingOutputValueMin	:REAL;			(* min Scaling Value on Output *)
	ScalingOutputValueMax	:REAL;			(* max Scaling Value on Output *)

END_STRUCT
END_TYPE

(* Data type in zLibrary/AnaIn *)
TYPE sAnaInVisu :
STRUCT
	InstName			:STRING(20);	(* Name of instance  *)
	Description			:STRING(32);	(* Description  *)
	BitInName			:STRING(25);	(* Name of bit input  *)

(* Outputvariables *)
	State				:DINT;			(* State of the outinput check *)
	AnaInValue			:REAL;
	HomePosition		:BOOL;			(* Object in home position  *)
	ErrorString			:STRING(40);	(* string shows missing signal *)
	ErrorPresent			: BOOL;
END_STRUCT
END_TYPE

(* Data type in zLibrary/AnaIn *)
TYPE sEncoderInit :
STRUCT
	InstName				:STRING(20);	(* Name of instance  *)
	Description				:STRING(32);	(* Description  *)
	BitInName				:STRING(25);	(* Name of bit input *)

	lr_LaengeProRpm			:LREAL;			(* mm *)
	i_InkProRpm				:UDINT		:=1440;		(*360 * 4*)	(* Inkremente pro Umdehung *)
END_STRUCT
END_TYPE

(* Data type in zLibrary/AnaIn *)
TYPE sEncoderVisu :
STRUCT
	InstName			:STRING(20);	(* Name of instance  *)
	Description			:STRING(32);	(* Description  *)
	BitInName			:STRING(25);	(* Name of bit input  *)

	Reset				:BOOL;

(* Outputvariables *)
	State				:DINT;			(* State of the outinput check *)
	ErrorString			:STRING(40);	(* string shows missing signal *)
	ErrorPresent			: BOOL;
	Drehrichtung		:enum_Drehrichtung;
	rpmValue			:LREAL;			(* rpm *)
	posValue			:LREAL;			(* mm *)
END_STRUCT
END_TYPE

(* Data type in zLibrary/CSV_Handling *)
TYPE CSV_Config :
STRUCT
	ColName				:STRING(30);
	ColDataType			:INT;
	ColSourceAdr		:DWORD;
	ColSourceSize		:DWORD;

END_STRUCT
END_TYPE

(* Data type in zLibrary/CSV_Handling *)
TYPE DataTypeDef :
STRUCT

	iBOOL		:INT:=1;
	iBYTE		:INT:=2;
	iWORD		:INT:=3;
	iDWORD		:INT:=4;
	iSINT		:INT:=5;
	iUSINT		:INT:=6;
	iINT		:INT:=7;
	iUINT		:INT:=8;
	iDINT		:INT:=9;
	iUDINT		:INT:=10;
	iREAL		:INT:=11;
	iLREAL		:INT:=12;
	iSTRING		:INT:=13;
	iTIME		:INT:=14;
	iTOD		:INT:=15;
	iDATE		:INT:=16;
	iDT			:INT:=17;

END_STRUCT
END_TYPE

(* Data type in zLibrary/DigIn *)
TYPE sDigInInit :
STRUCT
	InstName			: STRING(25);		(* Name of instance  *)
	Description			: STRING(50);		(* Description  *)
	BitInName			: STRING(25);		(* Name of bit input *)
	HomePosSignal		: DINT;				(* home-position is definded if : 0: Signal=Low, 1: Signal=High, 2: always  *)
	MaxTime				: DINT; 			(* number in ms cycles to Timeout *)
	EnableInEveryMode	: BOOL;				(* Object can be Controlled in every Mode *)

	IputOnDelayTime		: DINT;				(* number in ms for On - Delay SignalInDelayed *)
	IputOffDelayTime	: DINT;				(* number in ms for On - Delay SignalInDelayed *)

END_STRUCT
END_TYPE

(* Data type in zLibrary/DigIn *)
TYPE sDigInVisu :
STRUCT
	InstName				: STRING(25);		(* string shows instance name *)
	Description				: STRING(50);		(* Description        *)
	BitInName				: STRING(25);		(* Name of bit input  *)

(* Inputvariables *)
	BtnReset				: sButtonVisu;		(* Manage button *)

(* Outputvariables *)
	State					: StateObject;			(* State of the outinput check *)
	HomePosition			: BOOL;					(* Object in home position  *)
	ErrorString				: STRING(40);			(* string shows missing signal *)
	ErrorPresent			: BOOL;

(* Internal variables *)
	BitInToCheck			: BOOL;					(* Bit input signal  *)
	ProcessTime				: DINT;					(* Counts the time in ms						*)
	BtnResetVisible			: BOOL;					(* Switch for reset the input check *)

END_STRUCT
END_TYPE

(* Data type in zLibrary/DigOutIn *)
TYPE sDigOutInHome :
(
	HOME_LOW			:=0,
	HOME_HIGH 			:=1,
	HOME_NOT_DEFINED 	:=2

);
END_TYPE

(* Data type in zLibrary/DigOutIn *)
TYPE sDigOutInInit :
STRUCT
	InstName				: STRING(25);	(* Name of instance  *)
	Description				: STRING(50);	(* Description  *)

	BitOutName				: STRING(25);	(* Name of bit output*)
	BitInName				: STRING(25);	(* Name of bit input *)
	HomePosSignal			: DINT;			(* home-position is definded if :
															 	0: Signal=Low, 1: Signal=High, 2: always  *)
	HomePosOutput			: DINT;			(* home-position is definded if :
															 	0: Output=Low, 1: Output=High, 2: always  *)
	MaxTime					: DINT; 			(* number in ms cycles to Timeout *)
	EnableInEveryMode		: BOOL;			(* Object can be Controlled in every Mode *)
	EnableVisuInEveryMode	: BOOL;			(* Object can be Controlled from Visu in every Mode *)

END_STRUCT
END_TYPE

(* Data type in zLibrary/DigOutIn *)
TYPE sDigOutInVisu :
STRUCT
	InstName				:STRING(25);	(* string shows instance name *)
	Description				:STRING(50);	(* Description        *)
	BitOutName				:STRING(25);	(* Name of bit output *)
	BitInName				:STRING(25);	(* Name of bit input *)

(* Inputvariables *)
	BtnOutput				:sButtonVisu;	(* Manage button *)

(* Outputvariables *)
	State					:StateObject;	(* State of the outinput check *)
	OutputAvailable			:BOOL;			(* Output available *)
	InputAvailable			:BOOL;			(* Input available 	*)
	HomePosition			:BOOL;			(* Object in home position  *)
	ErrorString				:STRING(40);	(* string shows missing signal *)
	ErrorPresent			: BOOL;

(* Internal variables *)
	BitOutToSet				:BOOL;			(* Bit output signal *)
	BitInToCheck			:BOOL;			(* Bit input signal  *)
	ProcessTime				:DINT;			(* Counts the time in ms *)
	BtnResetVisible			:BOOL;			(* Switch for reset the input check *)
END_STRUCT
END_TYPE

(* Data type in zLibrary/EsponRobot/Drives_IO *)
TYPE sSMCGlobalVar :
STRUCT
 ObjCount			: INT 					:=0;
END_STRUCT
END_TYPE

(* Data type in zLibrary/EsponRobot/Drives_IO *)
TYPE sSMCInit :
STRUCT
	InstName					:	STRING(20);	(* Instance name of the object *)
	Description				:	STRING(50);	(* Description of instance     *)
	MaxTime						:	DINT; 			(* number of 100ms cycles to Timeout *)
	StepDataFilePath	:	STRING(80);	(* path for pos. file from ACT Controller export *)
END_STRUCT
END_TYPE

(* Data type in zLibrary/EsponRobot/Drives_IO *)
TYPE sSMCPosStruct :
STRUCT
	MoveFct 					:	STRING(8);
	PosValue  				:	REAL;
END_STRUCT
END_TYPE

(* Data type in zLibrary/EsponRobot/Drives_IO *)
TYPE sSMCVisu :
STRUCT
(* EA's from Axis *)
	In_Busy           : BOOL;
	In_Area           : BOOL;
	In_SetupOk        : BOOL;
	In_InPosition     : BOOL;
	In_Ready          : BOOL;
	In_EstopOk        : BOOL;
	In_NoAlarm        : BOOL;
	qRelease          : BOOL;
	qStepDataNo_0     : BOOL;
	qStepDataNo_1     : BOOL;
	qStepDataNo_2     : BOOL;
	qStepDataNo_3     : BOOL;
	qStepDataNo_4     : BOOL;
	qStepDataNo_5     : BOOL;
	qSetup            : BOOL;
	qMoveHold         : BOOL;
	qMoveStart        : BOOL;
	qReset            : BOOL;
	qServoOn          : BOOL;

(* Outputvariables*)
	State								: DINT;					(* State of the valve												*)
	HomePosition				: BOOL; 				(* valve in home-position										*)
	ErrorString					: STRING(40);		(* string shows missing signal 							*)
	InstName						:	STRING(20);		(* Instance name of the object *)
	Description					:	STRING(40);		(* Description of instance     *)
	ProcessTime					: DINT;					(* Process time *)
	PosArray						: ARRAY [0..63] OF sSMCPosStruct;
	ShowPosArray				: BOOL;

(* From Visu to Object *)
	PosNo								:	DINT;					(* Position No from Robot *)

	BtnRelease					:	sButtonVisu;	(* Manage button *)
	BtnSetup						:	sButtonVisu;	(* Manage button *)
	BtnMoveHold					:	sButtonVisu;	(* Manage button *)
	BtnMoveStart				:	sButtonVisu;	(* Manage button *)
	BtnReset    				:	sButtonVisu;	(* Manage button *)
	BtnServoOn  				:	sButtonVisu;	(* Manage button *)
	BtnReadFile  				:	sButtonVisu;	(* Manage button *)
END_STRUCT
END_TYPE

(* Data type in zLibrary/EsponRobot *)
TYPE sEpsonRobotInit :
STRUCT
(* Structure for initialising a valve *)
	BitName				: STRING(20);	(* Name of bit *)
	InstName			: STRING(20);	(* Instance name of the object *)
	Description			: STRING(50);	(* Description of instance *)

	MaxTime				: DINT; 			(* number of 100ms cycles to Timeout *)
	TcpIPSocket			: DINT; 			(* Socket No of TCP-IP Connection *)
	TcpIPAdress			: STRING(16); 	(* IP-Adress of TCP-IP Connection *)
	WithToolHandling	: BOOL;
	ToolMaxTime			: DINT;

END_STRUCT
END_TYPE

(* Data type in zLibrary/EsponRobot *)
TYPE sEpsonRobotRecvData :
STRUCT
	Alive			: DINT;
	TelNo			: DINT;
	PosNo			: DINT;
	PosX			: REAL;
	PosY			: REAL;
	PosZ			: REAL;
	ApplPara		: ARRAY[0..7] OF	REAL;
	ErrorCode		: DINT;

END_STRUCT
END_TYPE

(* Data type in zLibrary/EsponRobot *)
TYPE sEpsonRobotSendData :
STRUCT
	Alive			:	DINT;
	TelNo			:	DINT;
	PosNo			:	DINT;
	Override	:	DINT;
	Vel				:	DINT;
	Acc				:	DINT;
	OffsetX			:	REAL;
	OffsetY			:	REAL;
	OffsetZ			:	REAL;
	ApplPara	:	ARRAY[0..7] OF	REAL;

END_STRUCT
END_TYPE

(* Data type in zLibrary/EsponRobot *)
TYPE sEpsonRobotToolSettings :
STRUCT
(* Structure for initialising robot tool *)
	NameCoilA			: STRING(20);
	NameCoilB			: STRING(20);
	NameInitSensor		: STRING(20);
	NameWorkSensor	: STRING(20);
	NameBtnToolOn		: STRING(30);
	NameBtnToolOff		: STRING(30);
END_STRUCT
END_TYPE

(* Data type in zLibrary/EsponRobot *)
TYPE sEpsonRobotVisu :
STRUCT
(* Structure for Handshake to display a Epson Robot *)
(*--------------------------------------------------------------*)
(* sInit-Datas *)
	BitName					: STRING(20);	(* Name of bit *)
	InstName					: STRING(20);	(* Instance name of the object *)
	Description					: STRING(50);	(* Description of instance *)
	TcpIpAdress				: STRING(15);
	SocketState 				: STRING(20);

(* sRobotToolSetting-Datas *)
	WithToolHandling			: BOOL;
	NameCoilA					: STRING(20);
	NameCoilB					: STRING(20);
	NameInitSensor				: STRING(20);
	NameWorkSensor			: STRING(20);

(* Outputvariables*)
	State						: StateObject;	(* State of the valve*)
	HomePosition				: BOOL; 		(* valve in home-position*)
	ErrorString					: STRING(80);	(* string shows missing signal*)
	ErrorPresent					: BOOL;
	ActualPosition				: DINT;
	ActualArea					: DINT;
	ConnectionAlive				: BOOL;
	PosX						: REAL;
	PosY						: REAL;
	PosZ						: REAL;
	PosArray					: ARRAY[1..20] OF STRING(30);

(* From Visu to Object *)
	PosNo						: DINT;			(* Position No from Robot *)
	OffsetX						: REAL;			(* Offset X *)
	OffsetY						: REAL;			(* Offset Y *)
	OffsetZ						: REAL;			(* Offset Z *)
	ApplPara					: ARRAY[0..7] OF REAL; (* Machinespecific Values *)

(* Internal Variables*)
	ProcessTime				: DINT;			(* Counts the time in ms*)
	PosOffset					: DINT;

	BtnMove					: sButtonVisu;	(* Manage button *)
	BtnReset					: sButtonVisu;	(* Manage button *)
	BtnPrgStart					: sButtonVisu;	(* Manage button *)
	BtnPrgStop					: sButtonVisu;	(* Manage button *)
	BtnToolOn 					: sButtonVisu;	(* Manage button *)
	BtnToolOff					: sButtonVisu;	(* Manage button *)

(* Internal Variables used only in Visu *)
	ShowDetails					: BOOL;
	ShowPosArray				: BOOL;

(* EA's from Robot *)
	RemOutStart				: BOOL; 		(* For Moving to WorkPosition *)
	RemOutStop				: BOOL; 		(* For Moving to WorkPosition *)
	RemOutPause				: BOOL; 		(* For Moving to WorkPosition *)
	RemOutCont				: BOOL; 		(* For Moving to WorkPosition *)
	RemOutReset				: BOOL; 		(* For Moving to WorkPosition *)
	RemOutPowerOn			: BOOL; 		(* For Moving to WorkPosition *)
	RemOutPowerOff			: BOOL; 		(* For Moving to WorkPosition *)
	RemOutPowerHi				: BOOL; 		(* For Moving to WorkPosition *)
	RemOutSetToolOn			: BOOL; 		(* Anforderung Ausgang Robotertool EIN *)
	RemOutSetToolOff			: BOOL; 		(* Anforderung Ausgang Robotertool AUS *)

	RemInReady				: BOOL; 		(* For Moving to WorkPosition *)
	RemInRunning				: BOOL; 		(* For Moving to WorkPosition *)
	RemInPaused				: BOOL; 		(* For Moving to WorkPosition *)
	RemInError					: BOOL; 		(* For Moving to WorkPosition *)
	RemInEStopOn				: BOOL; 		(* For Moving to WorkPosition *)
	RemInSafeguardOn			: BOOL; 		(* For Moving to WorkPosition *)
	RemInSError				: BOOL; 		(* For Moving to WorkPosition *)
	RemInWarning				: BOOL; 		(* For Moving to WorkPosition *)

	RemInTcpIP_Wait			: BOOL; 		(* For Moving to WorkPosition *)
	RemInAreaBit1				: BOOL; 		(* For Moving to WorkPosition *)
	RemInAreaBit2				: BOOL; 		(* For Moving to WorkPosition *)
	RemInAreaBit4				: BOOL; 		(* For Moving to WorkPosition *)

	RemInToolCoilA				: BOOL;			(* Rückmeldung Tool CoilA/ Ausgang 1 ist ein *)
	RemInToolCoilB				: BOOL;			(* Rückmeldung Tool CoilB/ Ausgang 2 ist ein *)
	RemInToolInitSensor			: BOOL;			(* Tool Ruhesensor *)
	RemInToolWorkSensor		: BOOL;			(* Tool Ruhesensor *)

END_STRUCT
END_TYPE

(* Data type in zLibrary/KeyenceEtherCat *)
TYPE st_config_Keyence :
STRUCT
	Description				:STRING;
	InstName				:STRING;
	Aktiv					:BOOL;
END_STRUCT
END_TYPE

(* Data type in zLibrary/KeyenceEtherCat *)
TYPE st_ctrl_out_Keyence :
STRUCT
			iJobNo					:INT;

(*Bit 0*)	bReset					:BOOL;	(*Reserviert (alles zurücksetzen)*)
(*Bit 1*)	bPrgChange				:BOOL;	(*Programmwechselanforderung*)
(*Bit 2*)	bTrigger				:BOOL;	(*Trigger*)

(*nicht benutzt*)
(*Bit 3*) 	bMaster					:BOOL;	(*Master-Registrierunganforderung *)
(*Bit 4*) 	bSpeicherstopp			:BOOL;	(*Speicherstopp SD-Karte Anfrage*)
(*Bit 5*) 	bStatistikruecksetzung	:BOOL;	(* Statistikrücksetzung anfordern*)
(*Bit 6*) 	bFehlerLoeschen			:BOOL;	(*Anforderung Fehler löschen*)
(*Bit 7*) 	OCR_Seriennummer		:BOOL;	(*Anforderung OCR-Seriennummer Hochzählen*)
(*Bit 8*) 	Zaehlung_Ruecksetzen	:BOOL;	(*Zählung-Rücksetzen Anforderung*)
(*Bit 9*) 	Statistik_Ruecksetzen	:BOOL;	(*Anforderung Statistik aller Programme Rücksetzen*)
(*Bit 10*) 	Reserviert_10			:BOOL;	(**)
(*Bit 11*) 	Reserviert_11			:BOOL;	(**)
(*Bit 12*) 	Reserviert_12			:BOOL;	(**)
(*Bit 13*) 	Reserviert_13			:BOOL;	(**)
(*Bit 14*) 	Reserviert_14			:BOOL;	(**)
(*Bit 15*) 	Reserviert_15			:BOOL;	(**)


(*
DL-EC1A: PDO-Kommunikation (Prozessdaten-Objekte)

	Daten Senden via anInputRequest (* Index: 16#7000; SubIndex: 16#0001 - 16#0005 *)

	Index: 16#7000  SubIndex: 16#0001
		Inhalt:
			Bit 0 = Reserviert (alles zurücksetzen)
			Bit 1 = Programmwechselanforderung
			Bit 2 = Trigger
			Bit 3 = Master-Registrierunganforderung 
			Bit 4 = Speicherstopp SD-Karte Anfrage 
			Bit 5 = Statistikrücksetzung anfordern 
			Bit 6 = Anforderung Fehler löschen 
			Bit 7 = Anforderung OCR-Seriennummer Hochzählen 
			Bit 8 = Zählung-Rücksetzen Anforderung 
			Bit 9 = Anforderung Statistik aller Programme Rücksetzen
			Bit 10-15 = Reserviert
	Index: 16#7000  SubIndex: 16#0002
		Inhalt:
			Bit 0 = Reserviert	 (alles zurücksetzen)
			Bit 1 = Programmnummer ändern (Bit 0)
	Index: 16#7000  SubIndex: 16#0003
		Inhalt:
			Bit 0 = Reserviert  (alles zurücksetzen)
			Bit 1 = Programmnummer ändern (Bit 1)
	Index: 16#7000  SubIndex: 16#0004
		Inhalt:
			Bit 0 = Reserviert  (alles zurücksetzen)
			Bit 1 = Programmnummer ändern (Bit 2)
	Index: 16#7000  SubIndex: 16#0005
		Inhalt:
			Bit 0 = Reserviert
			Bit 1 = Programmnummer ändern (Bit 3)
*)

END_STRUCT
END_TYPE

(* Data type in zLibrary/Sensopart *)
TYPE eSensopartCommands:
	(
	Sensopart_Connect			:=10,
	Sensopart_Trigger			:=20
	);
END_TYPE

(* Data type in zLibrary/Valve *)
TYPE sValveGlobalVar :
STRUCT
 ObjCount			: INT 					:=0;
END_STRUCT
END_TYPE

(* Data type in zLibrary/Valve *)
TYPE sValveHome :
(
	HOME_INIT		:=0,
	HOME_WORK 	:=1,
	HOME_BOTH   :=2,
	HOME_ALWAYS :=3
);
END_TYPE

(* Data type in zLibrary/Valve *)
TYPE sValveInit :
STRUCT
(* Structure for initialising a valve *)
	BitName				: STRING(25);	(* Name of bit *)
	InstName				: STRING(25);	(* Instance name of the object *)
	Description				: STRING(50);	(* Description of instance     *)
	WorkDescription			: STRING;		(* Description of work movement for e.g. down	*)
	InitDescription			: STRING;		(* Description of init movement for e.g. up   *)

	KindOfValve				: STRING;		(* kind of the valve:				A, B, D, G*)
	HomePosDefine			: DINT;			(* home-position is definded in:			 				*)
																(* 0: InitPosition, 1: WorkPosition, 2: Both  *)
	MaxTime				: DINT; 			(* number of 100ms cycles to Timeout 				  *)
	DampBothTime			: DINT; 			(* time in msec. for damp both msec  					*)
	DisableSignalMonitoring 	: BOOL; 		(* Disable signalmonitoring after movement*)
END_STRUCT
END_TYPE

(* Data type in zLibrary/Valve *)
 TYPE sValveSensor_SensorOut :
STRUCT
	SensorName				:	STRING;	(* From Sensor: Sensorname *)
	SensorSignal			:	BOOL;		(* From Sensor *)
	SensorType				: sValveSensorType; (* From Sensor: Init- Or Worksensor *)
END_STRUCT
END_TYPE

(* Data type in zLibrary/Valve *)
 TYPE sValveSensor_ValveOut :
STRUCT
	SignalLoExpected	: BOOL; (* From Valve: If Sensor not Low Raise Error!  *)
	SignalHiExpected	: BOOL;	(* From Valve: If Sensor not High Raise Error!  *)
END_STRUCT
END_TYPE

(* Data type in zLibrary/Valve *)
TYPE sValveSensorInit :
STRUCT
(* Structure for initialising a valve *)
	BitName				: STRING(20);	(* Name of bit *)
	InstName				: STRING(20);	(* Instance name of the object *)
	Description				: STRING(50);	(* Description of instance     *)
	SensorType				: sValveSensorType;
END_STRUCT
END_TYPE

(* Data type in zLibrary/Valve *)
TYPE sValveSensorType :
(
	sValveSensorType_NotDefined		:=0,
	sValveSensorType_INIT					:=1,
	sValveSensorType_WORK 				:=2
);
END_TYPE

(* Data type in zLibrary/Valve *)
TYPE sValveVisu :
STRUCT
(* Structure for Handshake to display a valve *)
(*--------------------------------------------------------------*)
(* sInit-Datas *)
	BitName					: STRING(25);		(* Name of bit *)
	InstName				: STRING(25);		(* Instance name of the object *)
	Description				: STRING(50);		(* Description of instance     *)
	SAInitPosName			: STRING(16);		(* Name of Sensor Initpostion of cylinder A 	*)
	SAWorkPosName			: STRING(16);		(* Name of Sensor Workposition of cylinder A	*)
	SBInitPosName			: STRING(16);		(* Name of Sensor Initposition of cylinder B 	*)
	SBWorkPosName			: STRING(16);		(* Name of Sensor Workposition of cylinder B 	*)
	SCInitPosName			: STRING(16);		(* Name of Sensor Initposition of cylinder C 	*)
	SCWorkPosName			: STRING(16);		(* Name of Sensor Workposition of cylinder C 	*)
	SDInitPosName			: STRING(16);		(* Name of Sensor Initposition of cylinder D 	*)
	SDWorkPosName			: STRING(16);		(* Name of Sensor Workposition of cylinder D 	*)
	SEInitPosName			: STRING(16);		(* Name of Sensor Initposition of cylinder E 	*)
	SEWorkPosName			: STRING(16);		(* Name of Sensor Workposition of cylinder E 	*)
	WorkDescription			: STRING(16);		(* Description of work movement for e.g. down	*)
	InitDescription			: STRING(16);		(* Description of init movement for e.g. up   *)

	NoOfInitSensors			: DINT;				(* number of sensors in initposition:	0, 1 or 2, 3	*)
	NoOfWorkSensors			: DINT;				(* number of Sensors in workposition:	0, 1 or 2, 3	*)
	NoOfValveCoils			: DINT;				(* number of valvecoils:				1 or 2		*)
	KindOfValve				: STRING(4);		(* kind of the valve:				A, B, D, G, H or I  		*)
	HomePositionInfoNo 		: DINT;				(* missing to home position 									*)

(* Outputvariables*)
	State					: StateObject;		(* State of the valve*)
	HomePosition			: BOOL; 			(* valve in home-position*)
	ErrorString				: STRING(40);		(* string shows missing signal*)
	ErrorPresent			: BOOL;

(* Internal Variables*)
	AInitPosition			: BOOL; 			(* Sensor InitPosition of cylinder A*)
	AWorkPosition			: BOOL; 			(* Sensor WorkPosition of cylinder A*)
	BInitPosition			: BOOL; 			(* Sensor InitPosition of cylinder B*)
	BWorkPosition			: BOOL; 			(* Sensor WorkPosition of cylinder B*)
	CInitPosition			: BOOL; 			(* Sensor InitPosition of cylinder C*)
	CWorkPosition			: BOOL; 			(* Sensor WorkPosition of cylinder C*)
	DInitPosition			: BOOL; 			(* Sensor InitPosition of cylinder D*)
	DWorkPosition			: BOOL; 			(* Sensor WorkPosition of cylinder D*)
	EInitPosition			: BOOL; 			(* Sensor InitPosition of cylinder E*)
	EWorkPosition			: BOOL; 			(* Sensor WorkPosition of cylinder E*)
	CoilA					: BOOL; 			(* For Moving to WorkPosition*)
	CoilB					: BOOL; 			(* For Moving to InitPosition*)
	ProcessTime				: DINT;				(* Counts the time in ms*)

	BtnMoveWork				: sButtonVisu;		(* Manage button *)
	BtnMoveInit				: sButtonVisu;		(* Manage button *)
	BtnReset				: sButtonVisu;		(* Manage button *)

END_STRUCT
END_TYPE

(* POU pBasic/PLC_PRG, ST *)
PROGRAM PLC_PRG
VAR_OUTPUT
	GlobalHomePos		: BOOL;
END_VAR
VAR
	DW_alive			: DINT:=0;
	TimeStart			: TIME;
	TimeEnd				: TIME;
	fb_ton_startHYDRA	: TON;
END_VAR
DW_alive:=DW_alive+1;
TimeStart:=TIME();

BusDiagnosis();
(*LngHandler();*)
IOSimulation();
ErrorHandler.ClearAll(sVisu:=Visu.ErrorHandler);
MessageHandler.ClearAll(sVisu:=Visu.Message);
IF	ProcessMessage01 = '' OR ProcessMessage02 = '' OR
	ModeSelect.Mode<=MODE_MANUAL THEN
	ProcessMessage01:='EMPTY';
	ProcessMessage02:='EMPTY';
END_IF

ModeSelect(	sVisu				:=Visu.ModeSelect,
			ControlOn			:= ST00_200_A1_A1.BitInToCheck,
 			SafetyDoorOk		:= gReadyForControlOn,
			MainValveOk			:= ST00_350_B20_0.BitInToCheck OR		SpecialMode03.State=STATE_RUN(* @@@ *),
			EmergencyOk			:= ST00_200_A1_A1.BitInToCheck,
			BusControlState		:= STATE_OK,
			UserOK				:= TRUE,
			AutoCycleEnd 		:= CheckSFCInInit.AllSeqInInit,
			SpecialCycleEnd 	:= CallSpecialModeSFCs.AllSpecialModeSFCInInit,
			HomePosRunEnd 		:= PLC_PRG.GlobalHomePos AND HomePositionSFC.State=STATE_WAIT,
			AllDoorsClosed 		:= TRUE,
			EnableFromPrevMach	:= TRUE,
			EnableFromNextMach	:= TRUE,
			ProtecKeyNotIn		:= TRUE,
			ProtecNotBridged	:= TRUE,
			Enable 			    := TRUE,
			Reset 				:= FALSE,
					);

gResetAll:=ModeSelect.QReset;

CallGeneralFunctions();
(* Spezialfunktion: *)
(* Disconnect Scanner TCPIP-Gateway *)
gBasicManualMode:=ModeSelect.BasicManualMode;

(*----------------------------------------------------------------------------
 Main-Program
 ----------------------------------------------------------------------------*)

ST_UPS(b_Ups := TRUE);
ST_CPU();
ST_AutoCheckIn( i_IntervalDay:=7 );
ST_MainMenue();
ST_Path();
ST_MinExit();
ST_ReadXmlLine();
ST_ReadXmlLineMsg();
ST_SaveAndLoad();
ST_Lng();

fb_ton_startHYDRA(IN:=TD.ArtNo <> '',PT:=t#5s);
IF fb_ton_startHYDRA.Q THEN						(*Textdateien erst nach Einlesen der Typdaten (Maschinennummer>0) + 5 sekündiger Verzögerung schreiben/lesen*)

	(***Für HYDRA 8****************************************)
	ST_Hydra8();

	FbExportHydraString(s_Path:= 'C:\MPDV\AIP2\spool\',
					st_data:=st_Hydra8Data,
					s_system_time:=gVarStrSystemTime,
					sDateiName:= 'Eingang.txt',
					bKopiereDateiAufServer:=FALSE,
					sToolPath := s_tools_path,
					tStartTime:= T#5S);

	ST_ImportHydraString(s_Path:= 'C:\MPDV\AIP2\spool\',
						sDateiName:= 'Ausgang.txt',
						tStartTime := T#5S);

END_IF

IF gInitOk AND ST_Path.Done THEN

	ImpExp_UD(path:= s_ud_path,filename:='UserData.xml');

	UserLoginHandler(sVisu:= Visu.LoginHandler,UserList:=UD.UserList);
	TDHandler(TDActivationAlowed:= ModeSelect.Mode<=MODE_MANUAL ,sVisu:=sTDHandler);
	MPHandler(sVisu:=sMPHandler);
	MP_ShiftHandler();

	ListHomeNOK(Clear:=TRUE);
	gHomeOk:=TRUE;
	_CallFBs();

	GlobalHomePos:=gHomeOk (*AND gHomePosSFCDone*);


	_CallSFCs();
	_CallPRGs();
	CheckSFCInInit();

ELSE
	gInitCollect:=TRUE;
	_CallInit();
	gInitOk:=gInitCollect;
 (* Spezialfunktion: *)
END_IF (*gInitOk=TRUE*)

(*------------- Main-Program-End -------------------------------------------*)

ErrorHandler.HandleErrors(sVisu:=Visu.ErrorHandler);
ErrorHandler.VisuUpdate(sVisu:=Visu.ErrorHandler);
MessageHandler.VisuUpdate(sVisu:=Visu.Message);

TimeEnd:=TIME();

(*END Program -----------------------------------------------------------------*)
END_PROGRAM

(* POU System/BusDiagnosis/BusDiagnosis, ST *)
PROGRAM BusDiagnosis
VAR

	EtheCatMasterAmsNetId 		AT %I* 	: ARRAY[0..5] OF USINT;	(* AmsNetId of EtherCat Mater *)


	GetConfSlaves				: FB_EcGetConfSlaves;			(* Read all Configured Informations of Master *)
	GetScannedSlaves			: FB_EcGetScannedSlaves;
	GetAllSlaveStates			: FB_EcGetAllSlaveStates;

	ConfSlaveInfo 				: ARRAY[1..NoOfMaxSlaves] OF ST_EcSlaveConfigData;
	ScannedSlaveInfo 			: ARRAY[1..NoOfMaxSlaves] OF ST_EcSlaveScannedData;
	ScannedSlaveInfoTemp 		: ARRAY[1..NoOfMaxSlaves] OF ST_EcSlaveScannedData;

	SlaveStates					: ARRAY[1..NoOfMaxSlaves] OF ST_EcSlaveState;
	SlaveStatesTemp			: ARRAY[1..NoOfMaxSlaves] OF ST_EcSlaveState;
	StringSlaveStates			: ARRAY[1..NoOfMaxSlaves] OF STRING(80);


	FirstStart					: BOOL;

	WorkIdx					: DINT;
	ForIdx						: DINT;

END_VAR
VAR CONSTANT
	NoOfMaxSlaves				: DINT := 100;
END_VAR
(* Get EtherCat Config - ONCE after RESET *)
IF 	NOT FirstStart THEN
	GetConfSlaves.bExecute:=TRUE;
	FirstStart:=TRUE;
END_IF

(* Get actual EtherCat - Scan *)
CASE WorkIdx OF
0: (* Init *)
	WorkIdx:=1;
1: (* Start Getting Bus Scan *)
	GetScannedSlaves.bExecute:=TRUE;
	IF 	GetScannedSlaves.bBusy THEN
		WorkIdx:=2;
	END_IF
2:
	IF 	NOT GetScannedSlaves.bBusy THEN
		WorkIdx:=3;
		ScannedSlaveInfo:=ScannedSlaveInfoTemp;
	END_IF

3:(* Get Salve States *)
	GetAllSlaveStates.bExecute:=TRUE;
	IF 	GetAllSlaveStates.bBusy THEN
		WorkIdx:=4;
	END_IF
4:
	IF 	NOT GetAllSlaveStates.bBusy THEN
		WorkIdx:=5;
		SlaveStates:=SlaveStatesTemp;
		FOR ForIdx:=1 TO NoOfMaxSlaves DO
			StringSlaveStates[ForIdx]:=F_ConvSlaveStateToString(SlaveStates[ForIdx]);
		END_FOR
	END_IF
5: (* End of operation *)
	WorkIdx:=0;
END_CASE

GetConfSlaves(
	sNetId					:= GetAmsNetIdString(EtheCatMasterAmsNetId),
	pArrEcConfSlaveInfo		:= ADR(ConfSlaveInfo),
	cbBufLen				:= SIZEOF(ConfSlaveInfo),
);

GetConfSlaves.bExecute:=FALSE;

GetScannedSlaves(
	sNetId						:= GetAmsNetIdString(EtheCatMasterAmsNetId),
	pArrEcScannedSlaveInfo	:= ADR(ScannedSlaveInfoTemp),
	cbBufLen					:= SIZEOF(ScannedSlaveInfoTemp),
 );

GetScannedSlaves.bExecute:=FALSE;

GetAllSlaveStates(
	sNetId						:= GetAmsNetIdString(EtheCatMasterAmsNetId),
	pStateBuf					:= ADR(SlaveStatesTemp),
	cbBufLen					:= ADR(SlaveStatesTemp),
 );

GetAllSlaveStates.bExecute:=FALSE;
END_PROGRAM

(* POU System/BusDiagnosis/GetAmsNetIdString, ST *)
FUNCTION GetAmsNetIdString : STRING
VAR_INPUT
		EtheCatMasterAmsNetId : ARRAY[0..5] OF USINT;
END_VAR
VAR
	Idx : DINT;
END_VAR
GetAmsNetIdString:='';

FOR Idx:=0 TO 5 DO
	GetAmsNetIdString:=CONCAT(GetAmsNetIdString, USINT_TO_STRING(EtheCatMasterAmsNetId[Idx]));
	IF 	Idx<>5 THEN
		GetAmsNetIdString:=CONCAT(GetAmsNetIdString,'.');
	END_IF
END_FOR
END_FUNCTION

(* POU Stations/ST_00/ST00_PRGs/IOSimulation, ST *)
PROGRAM IOSimulation
VAR

END_VAR
SystemTaskInfoArr[1].cycleTimeExceeded;
SystemTaskInfoArr[1].lastExecTime;
END_PROGRAM

(* POU System/Error_and_Message/ErrorHandler, ST *)
PROGRAM ErrorHandler
VAR
	TempErrorArray					: sErrorHandlerVisu;
	TempErrorArrayLastCycle 		: sErrorHandlerVisu;
	TempErrorArrayLastCycleQuitt 	: sErrorHandlerVisu;
	Idx								: DINT;

	TempError						: BOOL;
	TempWarning					: BOOL;
	TempInfo						: BOOL;
	POS							: INT;
	i								: INT;

	(* Variable for ErrorHistory Handling *)
	Idx_Akt							: DINT;
	Idx_Last						: DINT;
	ErrorPresent						:BOOL;

	CompareValue					:DINT;

	(* Variables for ErrorLog.CSV *)
	ErrorLogBuffer				: ARRAY[0..100] OF ErrorStruct;
	EmptyError					: ErrorStruct;
	ErrorToLog					: ErrorStruct;
	ErrorToQuitt					: ErrorStruct;

	StepExportError				: DINT;

	(* CSV Config *)
	ColIdx						: DINT;
	DataType					: DataTypeDef;
	CSVConfig  					: ARRAY[1..20] OF CSV_Config;
	CSVConfigDone				: BOOL :=FALSE;
	ErrorExport					: CSVExport_AppendLineWithVarConfig;				(*Daten in CSV-Datei exportieren*)
END_VAR
VAR_INPUT
	ErrorLogFileName			: STRING(255) := ''; (* Filename with Path e.g. 'C:\ErrorLog.csv' *)
	ErrorToAdd					: ErrorStruct;
END_VAR
VAR_OUTPUT
	bOutError					: BOOL;
	bOutWarning				: BOOL;
	bOutInfo					: BOOL;
END_VAR
VAR_IN_OUT
	sVisu						: sErrorHandlerVisu;
END_VAR
;
END_PROGRAM
ACTION AddError:
FOR Idx:=0 TO NO_OF_ERRORS
DO

	IF TempErrorArray.Error[Idx].No=0
	THEN

		FOR i:=0 TO 5 DO	(*Leerstellen entfernen*)
			POS:=0;
			POS := FIND (ErrorToAdd.Text,'$R');
			IF POS <> 0 THEN
				ErrorToAdd.Text := DELETE (ErrorToAdd.Text,1,POS);
			END_IF
			POS:=0;
			POS := FIND (ErrorToAdd.Text,'$N');
			IF POS <> 0 THEN
				ErrorToAdd.Text := DELETE (ErrorToAdd.Text,1,POS);
			END_IF
		END_FOR

		TempErrorArray.Error[Idx]:=ErrorToAdd;
			CASE TempErrorArray.Error[Idx].Typ OF
				0: TempErrorArray.Error[Idx].LineColor:=color.salmon;
				1: TempErrorArray.Error[Idx].LineColor:=color.orange;
				2: TempErrorArray.Error[Idx].LineColor:=color.lightblue;
			END_CASE
		EXIT;
	END_IF
END_FOR
END_ACTION
ACTION ClearAll:
FOR Idx:=0 TO NO_OF_ERRORS
DO
	TempErrorArray.Error[Idx].No:=0;
	TempErrorArray.Error[Idx].No:=0;
	TempErrorArray.Error[Idx].DateTime:=DINT_TO_DT(0);
	TempErrorArray.Error[Idx].Text:='';
	TempErrorArray.Error[Idx].Typ:=0;
	TempErrorArray.Error[Idx].Station:=0;
	TempErrorArray.Error[Idx].Prio:=0;
	TempErrorArray.Error[Idx].QuitAddr:=0;
END_FOR
END_ACTION
ACTION HandleErrors:
TempError			:= FALSE;
TempWarning		:= FALSE;
TempInfo			:= FALSE;

FOR Idx:=0 TO NO_OF_ERRORS
DO
	IF TempErrorArray.Error[Idx].No<>0 AND TempErrorArray.Error[Idx].Typ=0 AND NOT TempError
	THEN
		TempError:=TRUE;
	END_IF
	IF TempErrorArray.Error[Idx].No<>0 AND TempErrorArray.Error[Idx].Typ=1 AND NOT TempWarning
	THEN
		TempWarning:=TRUE;
	END_IF
	IF TempErrorArray.Error[Idx].No<>0 AND TempErrorArray.Error[Idx].Typ=2 AND NOT TempInfo
	THEN
		TempInfo:=TRUE;
	END_IF
END_FOR

bOutError:=TempError;
bOutWarning:=TempWarning;
bOutInfo:=TempInfo;

(*Eintrag in die Errorlog, wenn der Fehler wieder weggeht-----------------------------------------------------------------------------------------------------------------*)
IF MEMCMP(ADR(TempErrorArray.Error), ADR(TempErrorArrayLastCycleQuitt.Error), SIZEOF(TempErrorArray.Error))<>0 THEN
	ErrorToQuitt:=EmptyError;
	FOR Idx_Akt:=0 TO NO_OF_ERRORS DO

		FOR Idx_Last:=0 TO NO_OF_ERRORS DO
			IF	(*TempErrorArrayLastCycleQuitt.Error[Idx_Akt].DateTime = TempErrorArray.Error[Idx_Last].DateTime AND*)
				TempErrorArrayLastCycleQuitt.Error[Idx_Akt].Text = TempErrorArray.Error[Idx_Last].Text OR
				(*Ausnahmen*)
				FIND(TempErrorArrayLastCycleQuitt.Error[Idx_Akt].Text, 'MessageHandler') >0 OR
				FIND(TempErrorArrayLastCycleQuitt.Error[Idx_Akt].Text, 'TD') >0 OR
				FIND(TempErrorArrayLastCycleQuitt.Error[Idx_Akt].Text, 'Mode') >0 OR
				FIND(TempErrorArrayLastCycleQuitt.Error[Idx_Akt].Text, 'LoginHandler') >0 THEN
				EXIT;
			END_IF
		END_FOR

		IF 	Idx_Last >NO_OF_ERRORS THEN
			ErrorToQuitt:=TempErrorArrayLastCycleQuitt.Error[Idx_Akt];
			ErrorToQuitt.DateTime:=gVarDTSystemtime;
			ErrorToQuitt.Text:=CONCAT('quitt ',ErrorToQuitt.Text);

			IF ErrorLogFileName<>'' THEN
				FOR Idx:= 100 TO 2 BY -1 DO
					ErrorLogBuffer[Idx]:=ErrorLogBuffer[Idx-1];
				END_FOR
				ErrorLogBuffer[1]:=ErrorToQuitt;
			END_IF
		END_IF

	END_FOR
END_IF
TempErrorArrayLastCycleQuitt:= TempErrorArray;
(*-------------------------------------------------------------------------------------------------------------------------------------------------------------------------------------------------------*)

(* Handle Error History *)

IF MEMCMP(ADR(TempErrorArray.Error), ADR(TempErrorArrayLastCycle.Error), SIZEOF(TempErrorArray.Error))<>0
THEN
	FOR Idx_Akt:=0 TO NO_OF_ERRORS
	DO
		ErrorPresent:=FALSE;
		FOR Idx_Last:=0 TO NO_OF_ERRORS
		DO
			CompareValue:=MEMCMP(ADR(TempErrorArray.Error[Idx_Akt].DateTime), ADR(TempErrorArrayLastCycle.Error[Idx_Last].DateTime), SIZEOF(TempErrorArray.Error[Idx_Akt].DateTime));
			IF TempErrorArray.Error[Idx_Akt].DateTime = TempErrorArrayLastCycle.Error[Idx_Last].DateTime
			THEN
				ErrorPresent:=TRUE;
				EXIT;
			END_IF
		END_FOR
		(* Error is not present in List *)
		IF NOT ErrorPresent AND TempErrorArray.Error[Idx_Akt].No<>0
		THEN
			(* Add To ErrorHistory *)
			FOR Idx:= 500 TO 2 BY -1
			DO
				ErrorHistory[Idx]:=ErrorHistory[Idx-1];
			END_FOR
			ErrorHistory[1]:=TempErrorArray.Error[Idx_Akt];
			(* Add To Error Log Buffer *)
			IF ErrorLogFileName<>''
				THEN
				FOR Idx:= 100 TO 2 BY -1
				DO
					ErrorLogBuffer[Idx]:=ErrorLogBuffer[Idx-1];
				END_FOR
				ErrorLogBuffer[1]:=TempErrorArray.Error[Idx_Akt];
			END_IF

		END_IF
	END_FOR
END_IF

TempErrorArrayLastCycle:= TempErrorArray;


IF visu.ErrorHistoryScroll>470 THEN
visu.ErrorHistoryScroll:=0;
END_IF

IF visu.ErrorHistoryScroll<0 THEN
visu.ErrorHistoryScroll:=0;
END_IF

FOR Idx:=0 TO NO_OF_ERRORS
DO
	IF	(Idx+visu.ErrorHistoryScroll) <= NO_OF_ERRORS THEN
		Visu.ErrorHistory.Error[Idx]:=ErrorHistory[Idx+visu.ErrorHistoryScroll];
		Visu.ErrorHistory.Error[Idx].No:=Idx+visu.ErrorHistoryScroll;
	END_IF
END_FOR

ErrorHandler.WriteErrorLog;
END_ACTION
ACTION VisuUpdate:
sVisu.Error:=TempErrorArray.Error;

(*
Das muss noch folgendermaßen umgesetzt werden.
(g.baiz, am 03.03.2010)

Das Visu-Array wird dem TempErrorArray abgeglichen,
d.h. für jeden Fehler wird "ObjektName" und "Fehlernummer" verglichen.

- Wenn Fehler noch in Visu aber nicht mehr in TempErrorArray, dann in Visu löschen
- Wenn Fehler bereits in Visu und noch im TempErrorArray, dann nur den "ErrorText" nochmals in die Visu kopieren 
  (könnte sich bei gleicher Fehlernummer geändert haben)
- Wenn Fehler noch nicht in Visu aber in TempErrorArray, dann Zeitstempel eintragen und in Visu kopieren

*)
END_ACTION
ACTION WriteErrorLog:
(* Config Log File *)
IF NOT CSVConfigDone
THEN
	ColIdx:=1;
	CSVConfig[ColIdx].ColName				:=	'Nr';
	CSVConfig[ColIdx].ColDataType		:=	DataType.iDINT;
	CSVConfig[ColIdx].ColSourceAdr		:=	ADR(ErrorToLog.No);
	CSVConfig[ColIdx].ColSourceSize	:=	SIZEOF(ErrorToLog.No);

	ColIdx:=ColIdx+1;
	CSVConfig[ColIdx].ColName				:=	'Datum/Uhrzeit';
	CSVConfig[ColIdx].ColDataType		:=	DataType.iDT;
	CSVConfig[ColIdx].ColSourceAdr		:=	ADR(ErrorToLog.DateTime);
	CSVConfig[ColIdx].ColSourceSize	:=	SIZEOF(ErrorToLog.DateTime);
	
	ColIdx:=ColIdx+1;
	CSVConfig[ColIdx].ColName				:=	'Beschreibung';
	CSVConfig[ColIdx].ColDataType		:=	DataType.iSTRING;
	CSVConfig[ColIdx].ColSourceAdr		:=	ADR(ErrorToLog.Text);
	CSVConfig[ColIdx].ColSourceSize	:=	SIZEOF(ErrorToLog.Text);
	
	ColIdx:=ColIdx+1;
	CSVConfig[ColIdx].ColName				:=	'Typ';
	CSVConfig[ColIdx].ColDataType		:=	DataType.iDINT;
	CSVConfig[ColIdx].ColSourceAdr		:=	ADR(ErrorToLog.Typ);
	CSVConfig[ColIdx].ColSourceSize	:=	SIZEOF(ErrorToLog.Typ);
	
	CSVConfigDone:=TRUE;
END_IF

(* Add To Error Log File *)
IF ErrorLogFileName<>''
THEN

	(* Check Error to Log present when Export inactive *)
	IF StepExportError = 0 THEN

		FOR Idx:= 1 TO 100
		DO
			IF ErrorLogBuffer[Idx].DateTime=EmptyError.DateTime
			THEN
				IF Idx>1
				THEN
					ErrorToLog:=ErrorLogBuffer[Idx-1];
					ErrorLogBuffer[Idx-1]:=EmptyError;
					StepExportError:=1;
				END_IF
				EXIT;
			END_IF
		END_FOR

	END_IF

	(* Export Error to specified CSV-File *)
	CASE StepExportError OF
	1: 	ErrorExport.nInExport:=TRUE;
		 	StepExportError:=2;
	2: 	IF ErrorExport.Done
			THEN
				StepExportError:=0;
			END_IF
	END_CASE

(* CylicCall *)
			ErrorExport(CSVConfig:=CSVConfig ,
									OverwriteExistingFile:=FALSE,
									strInFileName:=ErrorLogFileName ,
									localAMSNetID:= '',
									iInNumberOfColumns:= 4,
									CreateHeaderLine:=TRUE
									);

IF ErrorExport.Done
THEN
	ErrorExport.nInExport:=FALSE;
END_IF


END_IF
END_ACTION

(* POU zLibrary/CSV_ImportExport/CSVExport_AppendLineWithVarConfig, ST *)
FUNCTION_BLOCK CSVExport_AppendLineWithVarConfig
VAR_INPUT
	CSVConfig			: ARRAY[1..20] OF CSV_Config;
	nInExport			: BOOL;
	OverwriteExistingFile	: BOOL;
	strInFileName		: STRING(255);
	localAMSNetID		: T_AmsNetId;
	iInNumberOfColumns	: DINT;
	CreateHeaderLine	: BOOL;
END_VAR
VAR_OUTPUT
	Done				: BOOL;
END_VAR
VAR
	WorkingStep			: INT;
	WorkingStepWriteLine: INT;

	FindFile_			: FB_EnumFindFileEntry;
	filesList_			: ST_FindFileEntry;

